C07299=1019.054,-103.989,386.792,-23.976,21.681,-44.335
C07300=1019.057,-103.662,386.769,-23.976,21.681,-44.331
C07301=1019.060,-103.334,386.746,-23.977,21.680,-44.326
C07302=1019.062,-103.008,386.723,-23.978,21.680,-44.320
C07303=1019.065,-102.682,386.701,-23.978,21.679,-44.316
C07304=1019.067,-102.357,386.678,-23.979,21.679,-44.311
C07305=1019.070,-102.032,386.656,-23.980,21.678,-44.307
C07306=1019.072,-101.707,386.634,-23.980,21.677,-44.302
C07307=1019.075,-101.383,386.610,-23.981,21.677,-44.298
C07308=1019.077,-101.059,386.588,-23.981,21.676,-44.292
C07309=1019.079,-100.736,386.565,-23.982,21.676,-44.287
C07310=1019.082,-100.413,386.543,-23.983,21.675,-44.283
C07311=1019.085,-100.091,386.520,-23.983,21.675,-44.278
C07312=1019.086,-99.770,386.498,-23.984,21.674,-44.274
C07313=1019.089,-99.448,386.475,-23.985,21.673,-44.268
C07314=1019.091,-99.127,386.453,-23.985,21.673,-44.265
C07315=1019.094,-98.805,386.430,-23.986,21.673,-44.260
C07316=1019.096,-98.484,386.408,-23.986,21.671,-44.255
C07317=1019.099,-98.163,386.385,-23.987,21.672,-44.250
C07318=1019.101,-97.843,386.363,-23.987,21.670,-44.246
C07319=1019.103,-97.521,386.340,-23.988,21.670,-44.241
C07320=1019.106,-97.201,386.317,-23.989,21.670,-44.236
C07321=1019.108,-96.880,386.295,-23.989,21.669,-44.231
C07322=1019.110,-96.559,386.273,-23.990,21.669,-44.226
C07323=1019.112,-96.237,386.251,-23.991,21.668,-44.222
C07324=1019.114,-95.916,386.227,-23.991,21.668,-44.217
C07325=1019.116,-95.594,386.206,-23.992,21.667,-44.213
C07326=1019.118,-95.272,386.183,-23.993,21.666,-44.207
C07327=1019.121,-94.949,386.159,-23.993,21.666,-44.204
C07328=1019.123,-94.626,386.137,-23.994,21.666,-44.199
C07329=1019.125,-94.303,386.114,-23.994,21.665,-44.193
C07330=1019.127,-93.978,386.091,-23.995,21.664,-44.189
C07331=1019.129,-93.654,386.068,-23.996,21.664,-44.184
C07332=1019.131,-93.329,386.045,-23.996,21.663,-44.180
C07333=1019.133,-93.003,386.022,-23.997,21.663,-44.175
C07334=1019.135,-92.676,385.999,-23.998,21.662,-44.169
C07335=1019.138,-92.350,385.976,-23.998,21.662,-44.165
C07336=1019.140,-92.022,385.953,-23.999,21.661,-44.160
C07337=1019.142,-91.695,385.930,-23.999,21.660,-44.156
C07338=1019.144,-91.367,385.907,-24.000,21.660,-44.150
C07339=1019.146,-91.038,385.883,-24.001,21.660,-44.145
C07340=1019.148,-90.709,385.859,-24.001,21.659,-44.141
C07341=1019.150,-90.380,385.836,-24.002,21.658,-44.136
C07342=1019.152,-90.041,385.812,-24.003,21.658,-44.130
C07343=1019.154,-89.635,385.783,-24.004,21.657,-44.123
C07344=1019.156,-89.404,385.767,-24.004,21.656,-44.121
C07345=1019.157,-89.166,385.750,-24.004,21.656,-44.119
C07346=1019.159,-88.933,385.733,-24.004,21.656,-44.117
C07347=1019.159,-88.714,385.718,-24.005,21.656,-44.114
C07348=1019.162,-88.342,385.691,-24.006,21.655,-44.106
C07349=1019.164,-88.024,385.668,-24.006,21.654,-44.102
C07350=1019.166,-87.711,385.646,-24.007,21.654,-44.097
C07351=1019.167,-87.400,385.624,-24.007,21.653,-44.093
C07352=1019.169,-87.088,385.602,-24.008,21.653,-44.088
C07353=1019.171,-86.771,385.579,-24.009,21.652,-44.082
C07354=1019.173,-86.449,385.556,-24.009,21.652,-44.078
C07355=1019.174,-86.120,385.532,-24.010,21.651,-44.073
C07356=1019.177,-85.760,385.507,-24.011,21.650,-44.067
C07357=1019.178,-85.352,385.478,-24.012,21.649,-44.062
C07358=1019.180,-85.138,385.462,-24.012,21.649,-44.060
C07359=1019.181,-84.926,385.447,-24.012,21.650,-44.056
C07360=1019.183,-84.528,385.418,-24.013,21.649,-44.051
C07361=1019.185,-84.179,385.393,-24.014,21.648,-44.045
C07362=1019.187,-83.845,385.369,-24.015,21.648,-44.040
C07363=1019.188,-83.510,385.345,-24.015,21.647,-44.036
C07364=1019.190,-83.175,385.321,-24.016,21.647,-44.031
C07365=1019.192,-82.839,385.297,-24.016,21.646,-44.025
C07366=1019.194,-82.503,385.273,-24.017,21.645,-44.021
C07367=1019.194,-82.166,385.249,-24.018,21.645,-44.016
C07368=1019.197,-81.830,385.224,-24.018,21.645,-44.010
C07369=1019.198,-81.492,385.200,-24.019,21.644,-44.005
C07370=1019.200,-81.155,385.176,-24.020,21.643,-44.001
C07371=1019.202,-80.816,385.151,-24.020,21.643,-43.995
C07372=1019.203,-80.477,385.127,-24.021,21.643,-43.990
C07373=1019.205,-80.139,385.102,-24.021,21.641,-43.986
C07374=1019.206,-79.799,385.077,-24.022,21.641,-43.981
C07375=1019.208,-79.459,385.053,-24.023,21.641,-43.975
C07376=1019.210,-79.119,385.029,-24.023,21.639,-43.971
C07377=1019.211,-78.779,385.004,-24.024,21.639,-43.966
C07378=1019.212,-78.438,384.979,-24.025,21.638,-43.960
C07379=1019.214,-78.097,384.954,-24.026,21.639,-43.955
C07380=1019.215,-77.755,384.930,-24.026,21.637,-43.951
C07381=1019.217,-77.414,384.905,-24.027,21.637,-43.946
C07382=1019.218,-77.072,384.879,-24.028,21.636,-43.940
C07383=1019.220,-76.730,384.855,-24.028,21.636,-43.936
C07384=1019.221,-76.387,384.830,-24.029,21.635,-43.931
C07385=1019.223,-76.045,384.805,-24.030,21.635,-43.926
C07386=1019.224,-75.702,384.780,-24.030,21.634,-43.920
C07387=1019.225,-75.358,384.755,-24.031,21.634,-43.916
C07388=1019.226,-75.015,384.730,-24.031,21.633,-43.911
C07389=1019.228,-74.672,384.705,-24.032,21.633,-43.905
C07390=1019.230,-74.329,384.680,-24.033,21.632,-43.901
C07391=1019.231,-73.984,384.655,-24.033,21.632,-43.896
C07392=1019.232,-73.641,384.630,-24.034,21.631,-43.890
C07393=1019.233,-73.297,384.604,-24.035,21.630,-43.885
C07394=1019.235,-72.954,384.578,-24.035,21.630,-43.881
C07395=1019.236,-72.609,384.554,-24.036,21.629,-43.875
C07396=1019.237,-72.266,384.529,-24.037,21.629,-43.870
C07397=1019.238,-71.921,384.504,-24.038,21.628,-43.865
C07398=1019.240,-71.578,384.478,-24.038,21.628,-43.861
C07399=1019.241,-71.233,384.453,-24.039,21.627,-43.855
C07400=1019.242,-70.889,384.428,-24.040,21.627,-43.850
C07401=1019.243,-70.545,384.402,-24.040,21.626,-43.844
C07402=1019.244,-70.202,384.377,-24.041,21.625,-43.840
C07403=1019.246,-69.858,384.352,-24.041,21.625,-43.835
C07404=1019.246,-69.513,384.327,-24.042,21.624,-43.829
C07405=1019.248,-69.169,384.301,-24.043,21.624,-43.824
C07406=1019.249,-68.825,384.275,-24.043,21.623,-43.820
C07407=1019.249,-68.482,384.251,-24.044,21.623,-43.815
C07408=1019.251,-68.138,384.225,-24.045,21.622,-43.809
C07409=1019.252,-67.795,384.200,-24.045,21.622,-43.805
C07410=1019.253,-67.451,384.174,-24.046,21.621,-43.800
C07411=1019.254,-67.108,384.149,-24.047,21.621,-43.795
C07412=1019.255,-66.764,384.124,-24.048,21.620,-43.789
C07413=1019.256,-66.422,384.098,-24.048,21.620,-43.785
C07414=1019.257,-66.079,384.073,-24.049,21.619,-43.780
C07415=1019.258,-65.736,384.047,-24.050,21.619,-43.774
C07416=1019.259,-65.394,384.022,-24.050,21.617,-43.770
C07417=1019.260,-65.051,383.996,-24.051,21.618,-43.765
C07418=1019.261,-64.710,383.971,-24.051,21.617,-43.759
C07419=1019.262,-64.368,383.946,-24.052,21.617,-43.754
C07420=1019.262,-64.027,383.921,-24.053,21.615,-43.750
C07421=1019.264,-63.686,383.895,-24.053,21.616,-43.745
C07422=1019.264,-63.346,383.870,-24.054,21.615,-43.739
C07423=1019.265,-63.005,383.845,-24.055,21.614,-43.735
C07424=1019.266,-62.665,383.819,-24.055,21.613,-43.730
C07425=1019.266,-62.326,383.794,-24.056,21.614,-43.725
C07426=1019.267,-61.987,383.769,-24.057,21.612,-43.720
C07427=1019.268,-61.648,383.743,-24.057,21.612,-43.715
C07428=1019.269,-61.309,383.718,-24.058,21.611,-43.710
C07429=1019.270,-60.972,383.693,-24.059,21.611,-43.706
C07430=1019.270,-60.633,383.667,-24.059,21.610,-43.700
C07431=1019.271,-60.296,383.642,-24.060,21.610,-43.695
C07432=1019.272,-59.960,383.617,-24.060,21.609,-43.691
C07433=1019.272,-59.623,383.592,-24.061,21.609,-43.686
C07434=1019.272,-59.287,383.567,-24.062,21.608,-43.680
C07435=1019.274,-58.951,383.541,-24.062,21.608,-43.676
C07436=1019.274,-58.616,383.516,-24.063,21.607,-43.671
C07437=1019.275,-58.281,383.491,-24.064,21.607,-43.666
C07438=1019.276,-57.946,383.466,-24.064,21.606,-43.662
C07439=1019.276,-57.612,383.441,-24.065,21.606,-43.656
C07440=1019.276,-57.279,383.416,-24.066,21.605,-43.652
C07441=1019.277,-56.945,383.390,-24.066,21.604,-43.647
C07442=1019.277,-56.612,383.365,-24.067,21.605,-43.642
C07443=1019.279,-56.278,383.340,-24.068,21.603,-43.637
C07444=1019.278,-55.946,383.315,-24.068,21.603,-43.632
C07445=1019.279,-55.612,383.290,-24.069,21.603,-43.627
C07446=1019.280,-55.280,383.265,-24.070,21.602,-43.623
C07447=1019.280,-54.947,383.240,-24.070,21.602,-43.618
C07448=1019.281,-54.615,383.215,-24.071,21.601,-43.613
C07449=1019.281,-54.283,383.190,-24.072,21.601,-43.608
C07450=1019.281,-53.950,383.164,-24.072,21.600,-43.603
C07451=1019.282,-53.618,383.140,-24.073,21.599,-43.599
C07452=1019.282,-53.286,383.114,-24.074,21.600,-43.594
C07453=1019.283,-52.953,383.090,-24.074,21.598,-43.589
C07454=1019.283,-52.621,383.064,-24.075,21.598,-43.584
C07455=1019.283,-52.289,383.038,-24.075,21.597,-43.579
C07456=1019.284,-51.956,383.014,-24.076,21.597,-43.575
C07457=1019.284,-51.624,382.988,-24.077,21.597,-43.570
C07458=1019.284,-51.292,382.963,-24.077,21.596,-43.566
C07459=1019.285,-50.959,382.938,-24.078,21.596,-43.560
C07460=1019.285,-50.627,382.912,-24.079,21.595,-43.555
C07461=1019.285,-50.295,382.887,-24.079,21.594,-43.551
C07462=1019.285,-49.962,382.862,-24.080,21.595,-43.546
C07463=1019.285,-49.630,382.836,-24.080,21.593,-43.542
C07464=1019.286,-49.297,382.812,-24.081,21.593,-43.536
C07465=1019.286,-48.965,382.786,-24.081,21.592,-43.532
C07466=1019.287,-48.633,382.760,-24.082,21.592,-43.527
C07467=1019.286,-48.300,382.735,-24.083,21.592,-43.522
C07468=1019.287,-47.968,382.710,-24.083,21.591,-43.518
C07469=1019.287,-47.635,382.685,-24.084,21.591,-43.512
C07470=1019.287,-47.303,382.659,-24.085,21.589,-43.508
C07471=1019.287,-46.971,382.633,-24.086,21.589,-43.503
C07472=1019.287,-46.638,382.608,-24.086,21.590,-43.498
C07473=1019.287,-46.306,382.583,-24.087,21.588,-43.494
C07474=1019.287,-45.973,382.558,-24.088,21.588,-43.488
C07475=1019.287,-45.641,382.532,-24.088,21.588,-43.485
C07476=1019.288,-45.309,382.506,-24.089,21.587,-43.479
C07477=1019.287,-44.975,382.481,-24.089,21.586,-43.475
C07478=1019.288,-44.642,382.455,-24.090,21.586,-43.470
C07479=1019.288,-44.310,382.430,-24.091,21.586,-43.465
C07480=1019.288,-43.977,382.404,-24.091,21.585,-43.461
C07481=1019.288,-43.645,382.378,-24.092,21.585,-43.455
C07482=1019.287,-43.312,382.353,-24.092,21.584,-43.451
C07483=1019.287,-42.980,382.327,-24.093,21.583,-43.446
C07484=1019.288,-42.648,382.301,-24.094,21.583,-43.442
C07485=1019.288,-42.315,382.276,-24.094,21.583,-43.437
C07486=1019.287,-41.982,382.250,-24.095,21.582,-43.431
C07487=1019.287,-41.650,382.225,-24.096,21.582,-43.427
C07488=1019.286,-41.317,382.199,-24.096,21.582,-43.422
C07489=1019.287,-40.985,382.173,-24.097,21.580,-43.418
C07490=1019.287,-40.652,382.148,-24.098,21.580,-43.413
C07491=1019.287,-40.319,382.122,-24.098,21.580,-43.409
C07492=1019.287,-39.987,382.096,-24.099,21.579,-43.404
C07493=1019.286,-39.653,382.070,-24.100,21.579,-43.398
C07494=1019.286,-39.321,382.045,-24.100,21.578,-43.394
C07495=1019.286,-38.989,382.018,-24.101,21.578,-43.389
C07496=1019.286,-38.656,381.993,-24.101,21.577,-43.385
C07497=1019.285,-38.323,381.967,-24.102,21.577,-43.380
C07498=1019.285,-37.991,381.941,-24.102,21.576,-43.376
C07499=1019.285,-37.658,381.916,-24.103,21.576,-43.371
C07500=1019.285,-37.326,381.890,-24.104,21.575,-43.366
C07501=1019.284,-36.993,381.864,-24.105,21.575,-43.361
C07502=1019.284,-36.659,381.838,-24.105,21.574,-43.357
C07503=1019.284,-36.327,381.812,-24.106,21.574,-43.352
C07504=1019.284,-35.995,381.786,-24.107,21.574,-43.347
C07505=1019.283,-35.662,381.760,-24.107,21.573,-43.343
C07506=1019.283,-35.329,381.734,-24.108,21.573,-43.337
C07507=1019.283,-34.997,381.708,-24.108,21.572,-43.334
C07508=1019.282,-34.664,381.682,-24.109,21.572,-43.328
C07509=1019.281,-34.331,381.657,-24.109,21.571,-43.324
C07510=1019.281,-33.999,381.630,-24.110,21.571,-43.319
C07511=1019.281,-33.667,381.605,-24.111,21.570,-43.315
C07512=1019.280,-33.333,381.579,-24.111,21.570,-43.310
C07513=1019.280,-33.000,381.552,-24.112,21.569,-43.306
C07514=1019.280,-32.668,381.526,-24.113,21.569,-43.301
C07515=1019.279,-32.335,381.500,-24.113,21.568,-43.296
C07516=1019.279,-32.002,381.474,-24.114,21.568,-43.291
C07517=1019.278,-31.669,381.448,-24.114,21.567,-43.287
C07518=1019.278,-31.337,381.422,-24.115,21.567,-43.282
C07519=1019.277,-31.004,381.396,-24.116,21.566,-43.278
C07520=1019.276,-30.671,381.370,-24.116,21.566,-43.273
C07521=1019.276,-30.339,381.344,-24.117,21.565,-43.269
C07522=1019.275,-30.006,381.317,-24.118,21.565,-43.264
C07523=1019.274,-29.673,381.292,-24.118,21.565,-43.260
C07524=1019.275,-29.340,381.265,-24.119,21.564,-43.254
C07525=1019.274,-29.007,381.239,-24.119,21.563,-43.250
C07526=1019.273,-28.675,381.212,-24.120,21.563,-43.245
C07527=1019.273,-28.342,381.186,-24.120,21.562,-43.241
C07528=1019.272,-28.009,381.161,-24.121,21.562,-43.236
C07529=1019.271,-27.676,381.134,-24.122,21.562,-43.232
C07530=1019.270,-27.344,381.107,-24.123,21.562,-43.227
C07531=1019.270,-27.011,381.081,-24.123,21.560,-43.223
C07532=1019.269,-26.678,381.056,-24.124,21.560,-43.217
C07533=1019.269,-26.346,381.029,-24.124,21.560,-43.214
C07534=1019.267,-26.013,381.002,-24.125,21.559,-43.208
C07535=1019.267,-25.680,380.976,-24.126,21.559,-43.204
C07536=1019.266,-25.348,380.950,-24.126,21.559,-43.199
C07537=1019.265,-25.014,380.923,-24.127,21.558,-43.195
C07538=1019.265,-24.681,380.897,-24.128,21.558,-43.190
C07539=1019.264,-24.349,380.871,-24.128,21.557,-43.186
C07540=1019.263,-24.016,380.844,-24.129,21.557,-43.181
C07541=1019.263,-23.683,380.818,-24.129,21.556,-43.177
C07542=1019.262,-23.351,380.791,-24.130,21.556,-43.171
C07543=1019.260,-23.017,380.765,-24.131,21.555,-43.168
C07544=1019.260,-22.685,380.739,-24.131,21.556,-43.162
C07545=1019.259,-22.352,380.712,-24.132,21.554,-43.158
C07546=1019.258,-22.019,380.686,-24.133,21.554,-43.153
C07547=1019.257,-21.687,380.659,-24.133,21.554,-43.149
C07548=1019.256,-21.354,380.633,-24.134,21.553,-43.144
C07549=1019.255,-21.021,380.606,-24.134,21.552,-43.140
C07550=1019.254,-20.688,380.580,-24.135,21.553,-43.135
C07551=1019.253,-20.355,380.553,-24.136,21.552,-43.131
C07552=1019.253,-20.023,380.527,-24.136,21.551,-43.127
C07553=1019.251,-19.690,380.500,-24.137,21.551,-43.122
C07554=1019.251,-19.517,380.486,-24.137,21.550,-43.118
C07555=1019.250,-19.101,380.453,-24.138,21.550,-43.112
C07556=1019.249,-18.853,380.433,-24.139,21.550,-43.109
C07557=1019.248,-18.591,380.411,-24.139,21.550,-43.107
C07558=1019.248,-18.329,380.391,-24.139,21.549,-43.105
C07559=1019.247,-18.082,380.371,-24.139,21.548,-43.103
C07560=1019.246,-17.860,380.353,-24.140,21.549,-43.100
C07561=1019.245,-17.495,380.324,-24.141,21.548,-43.092
C07562=1019.244,-17.163,380.297,-24.141,21.547,-43.088
C07563=1019.243,-16.829,380.271,-24.142,21.547,-43.083
C07564=1019.241,-16.496,380.244,-24.142,21.547,-43.079
C07565=1019.240,-16.162,380.218,-24.143,21.546,-43.074
C07566=1019.240,-15.829,380.190,-24.144,21.546,-43.070
C07567=1019.238,-15.493,380.164,-24.145,21.546,-43.065
C07568=1019.237,-15.157,380.137,-24.145,21.545,-43.061
C07569=1019.236,-14.819,380.109,-24.146,21.544,-43.055
C07570=1019.235,-14.478,380.082,-24.146,21.544,-43.052
C07571=1019.233,-14.137,380.054,-24.147,21.544,-43.046
C07572=1019.232,-13.792,380.027,-24.147,21.543,-43.042
C07573=1019.231,-13.445,379.999,-24.148,21.543,-43.037
C07574=1019.230,-13.098,379.971,-24.149,21.542,-43.033
C07575=1019.228,-12.747,379.943,-24.149,21.542,-43.028
C07576=1019.227,-12.395,379.914,-24.150,21.541,-43.024
C07577=1019.226,-12.042,379.885,-24.151,21.541,-43.019
C07578=1019.224,-11.687,379.857,-24.151,21.540,-43.014
C07579=1019.223,-11.330,379.829,-24.152,21.540,-43.009
C07580=1019.222,-10.972,379.800,-24.152,21.539,-43.006
C07581=1019.220,-10.613,379.770,-24.153,21.539,-43.000
C07582=1019.219,-10.254,379.741,-24.154,21.539,-42.995
C07583=1019.217,-9.893,379.711,-24.154,21.538,-42.991
C07584=1019.216,-9.532,379.682,-24.155,21.538,-42.985
C07585=1019.215,-9.169,379.653,-24.156,21.537,-42.982
C07586=1019.213,-8.806,379.624,-24.156,21.536,-42.976
C07587=1019.212,-8.444,379.594,-24.157,21.536,-42.971
C07588=1019.210,-8.081,379.564,-24.158,21.536,-42.967
C07589=1019.208,-7.717,379.536,-24.158,21.535,-42.961
C07590=1019.206,-7.351,379.505,-24.159,21.535,-42.956
C07591=1019.205,-6.983,379.476,-24.160,21.534,-42.952
C07592=1019.203,-6.611,379.445,-24.160,21.534,-42.947
C07593=1019.201,-6.236,379.414,-24.161,21.533,-42.941
C07594=1019.199,-5.861,379.384,-24.162,21.533,-42.937
C07595=1019.198,-5.485,379.353,-24.163,21.533,-42.932
C07596=1019.196,-5.111,379.323,-24.163,21.532,-42.928
C07597=1019.194,-4.741,379.293,-24.164,21.532,-42.923
C07598=1019.193,-4.375,379.263,-24.164,21.531,-42.919
C07599=1019.191,-4.014,379.233,-24.165,21.530,-42.913
C07600=1019.189,-3.656,379.204,-24.166,21.531,-42.908
C07601=1019.187,-3.302,379.175,-24.166,21.529,-42.904
C07602=1019.186,-2.950,379.147,-24.167,21.529,-42.899
C07603=1019.184,-2.598,379.118,-24.167,21.529,-42.895
C07604=1019.183,-2.249,379.089,-24.168,21.529,-42.890
C07605=1019.181,-1.899,379.060,-24.169,21.528,-42.886
C07606=1019.179,-1.553,379.032,-24.169,21.528,-42.880
C07607=1019.177,-1.208,379.004,-24.170,21.527,-42.877
C07608=1019.175,-0.865,378.976,-24.170,21.527,-42.873
C07609=1019.174,-0.523,378.947,-24.171,21.526,-42.867
C07610=1019.172,-0.183,378.920,-24.172,21.526,-42.864
C07611=1019.170,0.155,378.892,-24.172,21.526,-42.858
C07612=1019.168,0.493,378.865,-24.173,21.525,-42.855
C07613=1019.166,0.828,378.837,-24.173,21.525,-42.851
C07614=1019.165,1.164,378.809,-24.174,21.525,-42.846
C07615=1019.163,1.497,378.782,-24.175,21.524,-42.842
C07616=1019.161,1.831,378.754,-24.175,21.523,-42.838
C07617=1019.160,2.161,378.727,-24.176,21.523,-42.834
C07618=1019.158,2.474,378.701,-24.176,21.523,-42.831
C07619=1019.155,2.762,378.678,-24.177,21.522,-42.827
C07620=1019.154,3.031,378.655,-24.177,21.522,-42.823
C07621=1019.152,3.292,378.633,-24.178,21.522,-42.818
C07622=1019.152,3.563,378.611,-24.179,21.521,-42.814
C07623=1019.150,3.852,378.588,-24.179,21.521,-42.810
C07624=1019.148,4.165,378.562,-24.179,21.520,-42.807
C07625=1019.146,4.495,378.535,-24.180,21.521,-42.803
C07626=1019.144,4.826,378.508,-24.180,21.519,-42.799
C07627=1019.142,5.157,378.479,-24.181,21.519,-42.795
C07628=1019.140,5.488,378.452,-24.181,21.518,-42.792
C07629=1019.139,5.818,378.425,-24.182,21.519,-42.786
C07630=1019.136,6.148,378.397,-24.183,21.518,-42.783
C07631=1019.135,6.478,378.370,-24.183,21.518,-42.779
C07632=1019.133,6.807,378.343,-24.184,21.518,-42.774
C07633=1019.131,7.135,378.316,-24.185,21.517,-42.770
C07634=1019.129,7.463,378.289,-24.185,21.517,-42.766
C07635=1019.126,7.788,378.262,-24.186,21.516,-42.762
C07636=1019.125,8.111,378.235,-24.186,21.516,-42.759
C07637=1019.122,8.432,378.208,-24.186,21.515,-42.755
C07638=1019.121,8.750,378.182,-24.187,21.516,-42.750
C07639=1019.119,9.067,378.156,-24.188,21.515,-42.746
C07640=1019.116,9.382,378.130,-24.188,21.515,-42.742
C07641=1019.115,9.697,378.104,-24.189,21.514,-42.738
C07642=1019.112,10.011,378.077,-24.190,21.514,-42.733
C07643=1019.110,10.327,378.051,-24.190,21.514,-42.730
C07644=1019.108,10.644,378.025,-24.191,21.513,-42.726
C07645=1019.106,10.963,377.998,-24.191,21.513,-42.722
C07646=1019.104,11.283,377.971,-24.192,21.512,-42.718
C07647=1019.102,11.605,377.944,-24.192,21.512,-42.715
C07648=1019.100,11.929,377.917,-24.193,21.511,-42.711
C07649=1019.098,12.253,377.891,-24.193,21.511,-42.707
C07650=1019.096,12.576,377.864,-24.194,21.511,-42.702
C07651=1019.093,12.899,377.836,-24.194,21.510,-42.698
C07652=1019.091,13.223,377.810,-24.195,21.510,-42.694
C07653=1019.089,13.547,377.782,-24.195,21.509,-42.691
C07654=1019.087,13.871,377.755,-24.196,21.509,-42.687
C07655=1019.084,14.195,377.729,-24.197,21.509,-42.682
C07656=1019.083,14.520,377.702,-24.197,21.509,-42.678
C07657=1019.080,14.845,377.674,-24.198,21.508,-42.674
C07658=1019.077,15.171,377.647,-24.198,21.508,-42.670
C07659=1019.076,15.496,377.620,-24.199,21.507,-42.667
C07660=1019.074,15.823,377.592,-24.199,21.507,-42.663
C07661=1019.070,16.150,377.565,-24.200,21.507,-42.658
C07662=1019.069,16.477,377.537,-24.200,21.506,-42.654
C07663=1019.066,16.805,377.510,-24.201,21.506,-42.650
C07664=1019.064,17.134,377.482,-24.201,21.505,-42.646
C07665=1019.061,17.464,377.455,-24.202,21.505,-42.643
C07666=1019.059,17.793,377.427,-24.202,21.504,-42.639
C07667=1019.056,18.124,377.399,-24.203,21.504,-42.634
C07668=1019.054,18.454,377.371,-24.204,21.504,-42.630
C07669=1019.051,18.786,377.343,-24.204,21.503,-42.626
C07670=1019.049,19.118,377.315,-24.205,21.503,-42.622
C07671=1019.047,19.449,377.288,-24.205,21.502,-42.619
C07672=1019.044,19.798,377.258,-24.206,21.503,-42.613
C07673=1019.041,20.215,377.223,-24.207,21.502,-42.608
C07674=1019.039,20.451,377.204,-24.207,21.502,-42.604
C07675=1019.037,20.698,377.182,-24.207,21.502,-42.603
C07676=1019.035,20.946,377.162,-24.208,21.502,-42.601
C07677=1019.033,21.188,377.141,-24.208,21.502,-42.599
C07678=1019.031,21.415,377.123,-24.208,21.501,-42.597
C07679=1019.029,21.622,377.105,-24.209,21.501,-42.593
C07680=1019.027,21.979,377.075,-24.209,21.500,-42.588
C07681=1019.025,22.303,377.047,-24.210,21.501,-42.584
C07682=1019.022,22.597,377.022,-24.210,21.500,-42.582
C07683=1019.020,22.850,377.001,-24.210,21.499,-42.580
C07684=1019.017,23.260,376.966,-24.211,21.499,-42.573
C07685=1019.014,23.668,376.932,-24.212,21.498,-42.565
C07686=1019.012,23.920,376.910,-24.213,21.498,-42.562
C07687=1019.009,24.214,376.886,-24.213,21.498,-42.560
C07688=1019.006,24.541,376.858,-24.213,21.497,-42.558
C07689=1019.004,24.875,376.830,-24.214,21.497,-42.553
C07690=1019.001,25.209,376.801,-24.215,21.497,-42.549
C07691=1018.998,25.544,376.773,-24.215,21.496,-42.545
C07692=1018.996,25.878,376.745,-24.216,21.496,-42.541
C07693=1018.992,26.212,376.717,-24.216,21.495,-42.538
C07694=1018.990,26.546,376.689,-24.217,21.495,-42.534
C07695=1018.987,26.881,376.659,-24.217,21.494,-42.530
C07696=1018.985,27.216,376.632,-24.218,21.494,-42.525
C07697=1018.982,27.549,376.603,-24.219,21.495,-42.522
C07698=1018.979,27.884,376.574,-24.219,21.494,-42.518
C07699=1018.976,28.219,376.546,-24.220,21.494,-42.514
C07700=1018.973,28.553,376.518,-24.220,21.493,-42.510
C07701=1018.970,28.887,376.490,-24.221,21.493,-42.507
C07702=1018.967,29.222,376.461,-24.221,21.492,-42.503
C07703=1018.965,29.556,376.432,-24.222,21.493,-42.498
C07704=1018.961,29.891,376.404,-24.222,21.492,-42.494
C07705=1018.959,30.225,376.376,-24.223,21.492,-42.490
C07706=1018.955,30.560,376.347,-24.223,21.491,-42.486
C07707=1018.953,30.895,376.318,-24.224,21.491,-42.483
C07708=1018.949,31.229,376.290,-24.224,21.490,-42.479
C07709=1018.947,31.563,376.262,-24.225,21.490,-42.475
C07710=1018.944,31.898,376.233,-24.225,21.489,-42.471
C07711=1018.941,32.233,376.204,-24.226,21.489,-42.468
C07712=1018.938,32.567,376.175,-24.226,21.489,-42.464
C07713=1018.934,32.902,376.147,-24.227,21.489,-42.459
C07714=1018.931,33.236,376.118,-24.228,21.489,-42.455
C07715=1018.928,33.571,376.090,-24.228,21.488,-42.452
C07716=1018.925,33.906,376.061,-24.229,21.488,-42.448
C07717=1018.922,34.241,376.033,-24.229,21.487,-42.444
C07718=1018.919,34.574,376.005,-24.230,21.487,-42.440
C07719=1018.916,34.909,375.976,-24.230,21.486,-42.437
C07720=1018.912,35.244,375.947,-24.231,21.486,-42.433
C07721=1018.910,35.579,375.918,-24.231,21.485,-42.429
C07722=1018.906,35.914,375.889,-24.232,21.486,-42.426
C07723=1018.903,36.248,375.861,-24.232,21.485,-42.422
C07724=1018.900,36.583,375.832,-24.233,21.485,-42.418
C07725=1018.897,36.917,375.803,-24.234,21.485,-42.413
C07726=1018.894,37.252,375.775,-24.234,21.485,-42.409
C07727=1018.891,37.587,375.746,-24.235,21.484,-42.405
C07728=1018.888,37.922,375.718,-24.235,21.484,-42.402
C07729=1018.884,38.257,375.688,-24.236,21.483,-42.398
C07730=1018.880,38.591,375.660,-24.236,21.483,-42.395
C07731=1018.877,38.926,375.631,-24.237,21.483,-42.391
C07732=1018.874,39.261,375.603,-24.237,21.483,-42.387
C07733=1018.871,39.596,375.573,-24.238,21.482,-42.383
C07734=1018.867,39.931,375.545,-24.238,21.482,-42.380
C07735=1018.865,40.265,375.516,-24.239,21.481,-42.376
C07736=1018.860,40.600,375.487,-24.239,21.481,-42.372
C07737=1018.857,40.934,375.458,-24.240,21.481,-42.369
C07738=1018.854,41.269,375.430,-24.240,21.481,-42.365
C07739=1018.850,41.604,375.400,-24.241,21.480,-42.361
C07740=1018.847,41.939,375.372,-24.241,21.480,-42.357
C07741=1018.844,42.274,375.344,-24.242,21.479,-42.354
C07742=1018.840,42.609,375.314,-24.242,21.479,-42.350
C07743=1018.837,42.944,375.286,-24.243,21.479,-42.347
C07744=1018.833,43.278,375.257,-24.243,21.479,-42.343
C07745=1018.830,43.614,375.228,-24.244,21.478,-42.339
C07746=1018.826,43.948,375.199,-24.244,21.478,-42.335
C07747=1018.823,44.284,375.170,-24.245,21.477,-42.332
C07748=1018.820,44.618,375.141,-24.245,21.477,-42.328
C07749=1018.816,44.953,375.112,-24.246,21.477,-42.325
C07750=1018.813,45.288,375.083,-24.246,21.477,-42.321
C07751=1018.809,45.624,375.054,-24.247,21.476,-42.317
C07752=1018.805,45.957,375.025,-24.247,21.476,-42.313
C07753=1018.801,46.293,374.996,-24.248,21.475,-42.309
C07754=1018.798,46.628,374.967,-24.248,21.475,-42.306
C07755=1018.795,46.963,374.938,-24.249,21.475,-42.302
C07756=1018.791,47.298,374.909,-24.249,21.475,-42.299
C07757=1018.787,47.633,374.880,-24.250,21.474,-42.295
C07758=1018.784,47.968,374.851,-24.250,21.474,-42.291
C07759=1018.780,48.302,374.822,-24.251,21.473,-42.287
C07760=1018.776,48.638,374.793,-24.251,21.473,-42.284
C07761=1018.772,48.973,374.764,-24.252,21.473,-42.280
C07762=1018.769,49.308,374.735,-24.252,21.473,-42.277
C07763=1018.765,49.642,374.706,-24.253,21.472,-42.273
C07764=1018.762,49.978,374.677,-24.253,21.472,-42.269
C07765=1018.758,50.313,374.647,-24.254,21.472,-42.266
C07766=1018.753,50.647,374.619,-24.254,21.471,-42.262
C07767=1018.750,50.983,374.590,-24.255,21.471,-42.258
C07768=1018.747,51.317,374.561,-24.255,21.471,-42.254
C07769=1018.743,51.653,374.532,-24.256,21.471,-42.251
C07770=1018.739,51.988,374.502,-24.256,21.470,-42.247
C07771=1018.735,52.323,374.473,-24.257,21.470,-42.244
C07772=1018.731,52.657,374.444,-24.257,21.470,-42.240
C07773=1018.727,52.993,374.415,-24.258,21.469,-42.238
C07774=1018.723,53.327,374.385,-24.258,21.469,-42.234
C07775=1018.720,53.663,374.357,-24.259,21.468,-42.230
C07776=1018.716,53.998,374.327,-24.259,21.468,-42.227
C07777=1018.711,54.332,374.298,-24.260,21.468,-42.223
C07778=1018.708,54.667,374.269,-24.260,21.468,-42.220
C07779=1018.704,55.003,374.240,-24.261,21.467,-42.216
C07780=1018.700,55.338,374.211,-24.261,21.467,-42.212
C07781=1018.696,55.673,374.181,-24.262,21.467,-42.209
C07782=1018.691,56.008,374.152,-24.262,21.467,-42.205
C07783=1018.688,56.343,374.123,-24.263,21.466,-42.201
C07784=1018.684,56.678,374.094,-24.263,21.466,-42.197
C07785=1018.680,57.013,374.064,-24.264,21.466,-42.194
C07786=1018.676,57.348,374.035,-24.264,21.465,-42.192
C07787=1018.672,57.682,374.006,-24.264,21.465,-42.188
C07788=1018.668,58.018,373.977,-24.265,21.464,-42.184
C07789=1018.664,58.353,373.947,-24.266,21.465,-42.181
C07790=1018.660,58.688,373.918,-24.266,21.464,-42.177
C07791=1018.656,59.022,373.889,-24.267,21.464,-42.173
C07792=1018.652,59.358,373.860,-24.267,21.464,-42.170
C07793=1018.647,59.693,373.829,-24.268,21.464,-42.166
C07794=1018.643,60.028,373.801,-24.268,21.463,-42.163
C07795=1018.639,60.363,373.771,-24.268,21.462,-42.160
C07796=1018.634,60.698,373.742,-24.269,21.462,-42.157
C07797=1018.631,61.033,373.712,-24.269,21.462,-42.153
C07798=1018.626,61.368,373.684,-24.270,21.461,-42.149
C07799=1018.622,61.703,373.653,-24.270,21.462,-42.146
C07800=1018.618,62.038,373.624,-24.271,21.461,-42.142
C07801=1018.614,62.372,373.595,-24.271,21.461,-42.139
C07802=1018.610,62.710,373.566,-24.272,21.460,-42.135
C07803=1018.604,63.106,373.531,-24.272,21.460,-42.131
C07804=1018.601,63.329,373.511,-24.273,21.461,-42.130
C07805=1018.600,63.547,373.491,-24.273,21.460,-42.128
C07806=1018.599,63.921,373.456,-24.274,21.460,-42.124
C07807=1018.598,64.278,373.423,-24.274,21.459,-42.120
C07808=1018.597,64.663,373.386,-24.274,21.459,-42.116
C07809=1018.596,65.059,373.349,-24.275,21.458,-42.113
C07810=1018.594,65.436,373.314,-24.276,21.459,-42.108
C07811=1018.594,65.790,373.280,-24.276,21.457,-42.105
C07812=1018.593,66.129,373.248,-24.277,21.458,-42.102
C07813=1018.592,66.462,373.216,-24.277,21.457,-42.098
C07814=1018.591,66.797,373.185,-24.278,21.457,-42.094
C07815=1018.590,67.134,373.153,-24.278,21.457,-42.091
C07816=1018.589,67.473,373.122,-24.279,21.457,-42.087
C07817=1018.588,67.811,373.089,-24.279,21.456,-42.085
C07818=1018.587,68.150,373.058,-24.279,21.456,-42.082
C07819=1018.587,68.490,373.025,-24.280,21.456,-42.078
C07820=1018.585,68.832,372.993,-24.280,21.455,-42.074
C07821=1018.584,69.173,372.960,-24.281,21.456,-42.071
C07822=1018.583,69.516,372.928,-24.281,21.455,-42.067
C07823=1018.582,69.860,372.896,-24.282,21.455,-42.063
C07824=1018.581,70.205,372.863,-24.282,21.454,-42.061
C07825=1018.580,70.550,372.830,-24.283,21.454,-42.058
C07826=1018.579,70.894,372.797,-24.283,21.453,-42.054
C07827=1018.578,71.238,372.765,-24.284,21.454,-42.051
C07828=1018.577,71.583,372.732,-24.284,21.453,-42.047
C07829=1018.576,71.928,372.699,-24.285,21.453,-42.043
C07830=1018.575,72.273,372.667,-24.285,21.453,-42.041
C07831=1018.574,72.619,372.633,-24.285,21.452,-42.037
C07832=1018.573,72.967,372.601,-24.286,21.452,-42.034
C07833=1018.572,73.317,372.567,-24.286,21.451,-42.030
C07834=1018.571,73.669,372.533,-24.287,21.452,-42.027
C07835=1018.570,74.022,372.500,-24.288,21.451,-42.023
C07836=1018.569,74.377,372.467,-24.288,21.451,-42.019
C07837=1018.568,74.734,372.432,-24.288,21.451,-42.017
C07838=1018.567,75.092,372.398,-24.289,21.450,-42.013
C07839=1018.566,75.449,372.364,-24.289,21.450,-42.010
C07840=1018.564,75.804,372.330,-24.290,21.450,-42.006
C07841=1018.563,76.151,372.297,-24.290,21.449,-42.004
C07842=1018.562,76.494,372.264,-24.291,21.449,-42.001
C07843=1018.562,76.830,372.232,-24.291,21.449,-41.997
C07844=1018.561,77.161,372.201,-24.292,21.449,-41.994
C07845=1018.559,77.487,372.169,-24.292,21.449,-41.990
C07846=1018.558,77.810,372.138,-24.292,21.448,-41.987
C07847=1018.558,78.134,372.108,-24.293,21.448,-41.984
C07848=1018.557,78.458,372.076,-24.293,21.448,-41.980
C07849=1018.555,78.786,372.045,-24.294,21.447,-41.977
C07850=1018.554,79.119,372.012,-24.295,21.448,-41.973
C07851=1018.553,79.457,371.980,-24.295,21.446,-41.971
C07852=1018.553,79.803,371.947,-24.295,21.447,-41.968
C07853=1018.551,80.154,371.914,-24.296,21.446,-41.964
C07854=1018.551,80.509,371.879,-24.296,21.446,-41.962
C07855=1018.549,80.865,371.845,-24.297,21.446,-41.958
C07856=1018.548,81.222,371.811,-24.297,21.445,-41.955
C07857=1018.546,81.578,371.776,-24.298,21.446,-41.951
C07858=1018.545,81.934,371.743,-24.298,21.445,-41.947
C07859=1018.544,82.288,371.708,-24.298,21.444,-41.945
C07860=1018.543,82.642,371.674,-24.299,21.444,-41.942
C07861=1018.542,82.995,371.641,-24.299,21.444,-41.938
C07862=1018.541,83.346,371.606,-24.300,21.444,-41.935
C07863=1018.540,83.697,371.573,-24.300,21.444,-41.931
C07864=1018.538,84.048,371.539,-24.301,21.443,-41.929
C07865=1018.537,84.396,371.505,-24.301,21.443,-41.925
C07866=1018.536,84.744,371.471,-24.302,21.443,-41.922
C07867=1018.536,85.091,371.438,-24.302,21.443,-41.918
C07868=1018.534,85.436,371.405,-24.302,21.442,-41.916
C07869=1018.534,85.780,371.371,-24.303,21.442,-41.912
C07870=1018.532,86.123,371.339,-24.303,21.442,-41.909
C07871=1018.531,86.465,371.305,-24.304,21.441,-41.906
C07872=1018.529,86.806,371.272,-24.304,21.441,-41.903
C07873=1018.529,87.146,371.240,-24.305,21.441,-41.899
C07874=1018.527,87.482,371.207,-24.305,21.441,-41.898
C07875=1018.526,87.815,371.174,-24.305,21.440,-41.894
C07876=1018.525,88.142,371.143,-24.306,21.441,-41.890
C07877=1018.524,88.464,371.112,-24.306,21.439,-41.888
C07878=1018.523,88.784,371.081,-24.307,21.440,-41.885
C07879=1018.522,89.105,371.049,-24.307,21.439,-41.881
C07880=1018.521,89.430,371.018,-24.308,21.439,-41.879
C07881=1018.520,89.759,370.986,-24.308,21.440,-41.876
C07882=1018.519,90.092,370.954,-24.308,21.438,-41.874
C07883=1018.518,90.427,370.921,-24.309,21.439,-41.870
C07884=1018.516,90.761,370.888,-24.309,21.438,-41.866
C07885=1018.516,91.095,370.856,-24.310,21.438,-41.865
C07886=1018.515,91.430,370.823,-24.310,21.438,-41.861
C07887=1018.513,91.765,370.791,-24.311,21.438,-41.857
C07888=1018.512,92.099,370.758,-24.311,21.437,-41.855
C07889=1018.510,92.433,370.726,-24.311,21.437,-41.852
C07890=1018.510,92.768,370.694,-24.312,21.436,-41.849
C07891=1018.509,93.102,370.660,-24.312,21.437,-41.846
C07892=1018.507,93.436,370.628,-24.313,21.436,-41.842
C07893=1018.506,93.771,370.595,-24.313,21.436,-41.841
C07894=1018.505,94.106,370.562,-24.314,21.436,-41.837
C07895=1018.504,94.440,370.530,-24.314,21.436,-41.833
C07896=1018.503,94.773,370.497,-24.314,21.436,-41.832
C07897=1018.502,95.108,370.465,-24.315,21.435,-41.828
C07898=1018.500,95.442,370.432,-24.315,21.435,-41.826
C07899=1018.499,95.777,370.399,-24.316,21.435,-41.822
C07900=1018.498,96.111,370.366,-24.316,21.435,-41.819
C07901=1018.497,96.445,370.334,-24.316,21.434,-41.817
C07902=1018.496,96.779,370.302,-24.317,21.434,-41.813
C07903=1018.495,97.114,370.268,-24.317,21.434,-41.811
C07904=1018.494,97.448,370.236,-24.318,21.434,-41.808
C07905=1018.492,97.782,370.203,-24.318,21.433,-41.806
C07906=1018.491,98.116,370.170,-24.318,21.433,-41.802
C07907=1018.490,98.450,370.138,-24.319,21.433,-41.799
C07908=1018.488,98.785,370.105,-24.319,21.432,-41.796
C07909=1018.488,99.119,370.071,-24.320,21.433,-41.793
C07910=1018.486,99.454,370.039,-24.320,21.432,-41.791
C07911=1018.485,99.787,370.006,-24.320,21.432,-41.787
C07912=1018.484,100.121,369.974,-24.321,21.432,-41.785
C07913=1018.483,100.455,369.941,-24.321,21.431,-41.782
C07914=1018.481,100.789,369.908,-24.322,21.432,-41.778
C07915=1018.481,101.124,369.875,-24.322,21.431,-41.776
C07916=1018.479,101.458,369.842,-24.323,21.431,-41.773
C07917=1018.478,101.792,369.809,-24.323,21.431,-41.771
C07918=1018.477,102.126,369.776,-24.323,21.430,-41.767
C07919=1018.476,102.460,369.743,-24.324,21.430,-41.765
C07920=1018.474,102.794,369.711,-24.324,21.431,-41.762
C07921=1018.473,103.128,369.677,-24.324,21.429,-41.760
C07922=1018.472,103.463,369.644,-24.325,21.430,-41.756
C07923=1018.471,103.797,369.611,-24.325,21.429,-41.752
C07924=1018.470,104.131,369.578,-24.326,21.429,-41.751
C07925=1018.468,104.465,369.546,-24.326,21.430,-41.747
C07926=1018.467,104.799,369.512,-24.326,21.428,-41.745
C07927=1018.465,105.133,369.480,-24.327,21.429,-41.742
C07928=1018.464,105.467,369.447,-24.327,21.428,-41.739
C07929=1018.464,105.801,369.413,-24.328,21.428,-41.736
C07930=1018.462,106.135,369.380,-24.328,21.428,-41.734
C07931=1018.461,106.469,369.347,-24.328,21.427,-41.730
C07932=1018.460,106.803,369.314,-24.329,21.427,-41.728
C07933=1018.458,107.137,369.282,-24.329,21.428,-41.725
C07934=1018.457,107.471,369.248,-24.329,21.427,-41.723
C07935=1018.456,107.805,369.215,-24.330,21.427,-41.719
C07936=1018.455,108.139,369.182,-24.330,21.427,-41.718
C07937=1018.454,108.473,369.149,-24.331,21.426,-41.714
C07938=1018.453,108.807,369.116,-24.331,21.426,-41.712
C07939=1018.452,109.141,369.083,-24.332,21.426,-41.708
C07940=1018.449,109.476,369.049,-24.332,21.425,-41.706
C07941=1018.448,109.809,369.016,-24.332,21.426,-41.703
C07942=1018.447,110.143,368.983,-24.333,21.425,-41.701
C07943=1018.446,110.477,368.949,-24.333,21.425,-41.697
C07944=1018.445,110.811,368.916,-24.333,21.425,-41.695
C07945=1018.444,111.145,368.883,-24.334,21.424,-41.692
C07946=1018.443,111.479,368.851,-24.334,21.424,-41.690
C07947=1018.441,111.813,368.817,-24.335,21.425,-41.686
C07948=1018.440,112.147,368.783,-24.335,21.423,-41.684
C07949=1018.438,112.481,368.750,-24.335,21.424,-41.681
C07950=1018.438,112.815,368.717,-24.336,21.424,-41.679
C07951=1018.437,113.149,368.683,-24.336,21.423,-41.675
C07952=1018.435,113.483,368.650,-24.336,21.423,-41.673
C07953=1018.434,113.817,368.618,-24.337,21.423,-41.670
C07954=1018.432,114.151,368.584,-24.337,21.422,-41.668
C07955=1018.431,114.485,368.551,-24.338,21.423,-41.664
C07956=1018.430,114.819,368.517,-24.338,21.422,-41.662
C07957=1018.429,115.153,368.484,-24.338,21.421,-41.660
C07958=1018.428,115.486,368.451,-24.339,21.422,-41.657
C07959=1018.426,115.821,368.417,-24.339,21.422,-41.655
C07960=1018.425,116.154,368.384,-24.340,21.422,-41.652
C07961=1018.424,116.488,368.350,-24.340,21.421,-41.649
C07962=1018.423,116.822,368.317,-24.340,21.421,-41.646
C07963=1018.421,117.156,368.283,-24.341,21.421,-41.644
C07964=1018.420,117.490,368.250,-24.341,21.421,-41.640
C07965=1018.419,117.824,368.217,-24.341,21.420,-41.638
C07966=1018.418,118.158,368.183,-24.342,21.421,-41.635
C07967=1018.416,118.492,368.149,-24.342,21.420,-41.633
C07968=1018.415,118.826,368.116,-24.342,21.419,-41.631
C07969=1018.414,119.160,368.083,-24.343,21.420,-41.628
C07970=1018.412,119.494,368.049,-24.343,21.419,-41.625
C07971=1018.411,119.828,368.016,-24.344,21.419,-41.622
C07972=1018.410,120.162,367.982,-24.344,21.419,-41.620
C07973=1018.408,120.496,367.948,-24.345,21.419,-41.617
C07974=1018.407,120.830,367.915,-24.345,21.418,-41.614
C07975=1018.406,121.163,367.882,-24.345,21.418,-41.613
C07976=1018.405,121.498,367.848,-24.346,21.418,-41.609
C07977=1018.403,121.832,367.814,-24.346,21.417,-41.607
C07978=1018.403,122.165,367.781,-24.346,21.418,-41.604
C07979=1018.401,122.499,367.747,-24.347,21.418,-41.602
C07980=1018.400,122.833,367.713,-24.347,21.418,-41.598
C07981=1018.398,123.167,367.679,-24.347,21.417,-41.596
C07982=1018.397,123.501,367.646,-24.348,21.417,-41.594
C07983=1018.396,123.836,367.613,-24.348,21.417,-41.591
C07984=1018.395,124.170,367.579,-24.348,21.417,-41.589
C07985=1018.393,124.503,367.545,-24.349,21.416,-41.585
C07986=1018.392,124.837,367.511,-24.349,21.416,-41.583
C07987=1018.391,125.171,367.477,-24.349,21.416,-41.581
C07988=1018.389,125.505,367.444,-24.350,21.416,-41.578
C07989=1018.388,125.839,367.410,-24.350,21.415,-41.576
C07990=1018.387,126.174,367.376,-24.351,21.416,-41.572
C07991=1018.386,126.507,367.343,-24.351,21.415,-41.571
C07992=1018.384,126.841,367.308,-24.351,21.415,-41.569
C07993=1018.383,127.175,367.275,-24.352,21.415,-41.565
C07994=1018.381,127.509,367.241,-24.352,21.415,-41.563
C07995=1018.381,127.844,367.207,-24.352,21.414,-41.561
C07996=1018.379,128.178,367.174,-24.353,21.415,-41.558
C07997=1018.378,128.511,367.140,-24.353,21.414,-41.555
C07998=1018.377,128.846,367.105,-24.354,21.414,-41.552
C07999=1018.376,129.179,367.072,-24.354,21.414,-41.550
C08000=1018.374,129.513,367.038,-24.354,21.414,-41.548
C08001=1018.373,129.847,367.004,-24.355,21.413,-41.545
C08002=1018.371,130.181,366.970,-24.355,21.413,-41.543
C08003=1018.370,130.516,366.936,-24.355,21.413,-41.541
C08004=1018.369,130.850,366.903,-24.356,21.413,-41.538
C08005=1018.368,131.184,366.868,-24.356,21.412,-41.535
C08006=1018.367,131.518,366.835,-24.356,21.412,-41.532
C08007=1018.365,131.852,366.801,-24.357,21.412,-41.530
C08008=1018.364,132.186,366.767,-24.357,21.412,-41.528
C08009=1018.363,132.520,366.733,-24.357,21.412,-41.525
C08010=1018.361,132.854,366.699,-24.358,21.411,-41.523
C08011=1018.360,133.189,366.665,-24.358,21.411,-41.521
C08012=1018.359,133.522,366.631,-24.358,21.411,-41.517
C08013=1018.358,133.857,366.596,-24.359,21.411,-41.515
C08014=1018.356,134.191,366.563,-24.359,21.410,-41.513
C08015=1018.356,134.525,366.528,-24.359,21.411,-41.510
C08016=1018.354,134.859,366.494,-24.360,21.410,-41.508
C08017=1018.352,135.193,366.460,-24.360,21.410,-41.506
C08018=1018.352,135.526,366.426,-24.361,21.411,-41.503
C08019=1018.350,135.849,366.393,-24.361,21.410,-41.501
C08020=1018.349,136.149,366.362,-24.361,21.410,-41.499
C08021=1018.348,136.429,366.334,-24.361,21.410,-41.497
C08022=1018.347,136.694,366.307,-24.361,21.409,-41.495
C08023=1018.345,136.958,366.280,-24.362,21.409,-41.491
C08024=1018.345,137.234,366.252,-24.362,21.409,-41.490
C08025=1018.344,137.532,366.221,-24.363,21.409,-41.488
C08026=1018.342,137.854,366.189,-24.363,21.408,-41.486
C08027=1018.342,138.194,366.154,-24.363,21.408,-41.484
C08028=1018.340,138.551,366.117,-24.364,21.408,-41.480
C08029=1018.338,138.962,366.075,-24.364,21.408,-41.477
C08030=1018.337,139.190,366.052,-24.364,21.408,-41.475
C08031=1018.337,139.427,366.027,-24.365,21.408,-41.473
C08032=1018.336,139.670,366.003,-24.365,21.408,-41.473
C08033=1018.335,139.911,365.977,-24.365,21.408,-41.471
C08034=1018.333,140.143,365.954,-24.365,21.408,-41.470
C08035=1018.332,140.364,365.931,-24.365,21.407,-41.469
C08036=1018.331,140.757,365.891,-24.366,21.407,-41.465
C08037=1018.330,141.102,365.856,-24.366,21.407,-41.462
C08038=1018.328,141.441,365.820,-24.367,21.407,-41.460
C08039=1018.328,141.781,365.786,-24.367,21.407,-41.457
C08040=1018.326,142.121,365.750,-24.367,21.406,-41.455
C08041=1018.325,142.462,365.716,-24.368,21.406,-41.453
C08042=1018.324,142.803,365.680,-24.368,21.407,-41.449
C08043=1018.323,143.145,365.646,-24.368,21.406,-41.448
C08044=1018.321,143.487,365.610,-24.369,21.405,-41.445
C08045=1018.320,143.831,365.574,-24.369,21.406,-41.442
C08046=1018.319,144.174,365.540,-24.369,21.405,-41.440
C08047=1018.317,144.518,365.504,-24.370,21.405,-41.438
C08048=1018.316,144.863,365.468,-24.370,21.406,-41.435
C08049=1018.315,145.208,365.433,-24.370,21.405,-41.432
C08050=1018.314,145.553,365.397,-24.371,21.404,-41.431
C08051=1018.312,145.898,365.362,-24.371,21.405,-41.427
C08052=1018.311,146.245,365.326,-24.371,21.405,-41.425
C08053=1018.309,146.590,365.291,-24.372,21.404,-41.424
C08054=1018.302,146.937,365.259,-24.372,21.404,-41.420
C08055=1018.283,147.282,365.234,-24.372,21.404,-41.418
C08056=1018.661,147.310,364.998,-24.372,21.404,-41.418
C08057=1018.682,146.965,365.022,-24.372,21.404,-41.420
C08058=1018.690,146.618,365.053,-24.372,21.404,-41.424
C08059=1018.692,146.272,365.088,-24.371,21.405,-41.425
C08060=1018.693,145.926,365.124,-24.371,21.405,-41.427
C08061=1018.695,145.581,365.161,-24.371,21.404,-41.431
C08062=1018.696,145.235,365.196,-24.370,21.405,-41.432
C08063=1018.697,144.890,365.231,-24.370,21.406,-41.435
C08064=1018.699,144.546,365.267,-24.370,21.405,-41.438
C08065=1018.699,144.201,365.302,-24.369,21.405,-41.440
C08066=1018.701,143.859,365.338,-24.369,21.406,-41.442
C08067=1018.702,143.515,365.373,-24.369,21.405,-41.445
C08068=1018.703,143.172,365.408,-24.368,21.406,-41.448
C08069=1018.705,142.831,365.443,-24.368,21.407,-41.449
C08070=1018.706,142.489,365.479,-24.368,21.406,-41.453
C08071=1018.707,142.149,365.514,-24.367,21.406,-41.455
C08072=1018.708,141.808,365.548,-24.367,21.407,-41.457
C08073=1018.710,141.468,365.583,-24.367,21.407,-41.460
C08074=1018.711,141.130,365.618,-24.366,21.407,-41.462
C08075=1018.712,140.785,365.654,-24.366,21.407,-41.465
C08076=1018.714,140.391,365.694,-24.365,21.407,-41.469
C08077=1018.715,140.171,365.717,-24.365,21.408,-41.470
C08078=1018.715,139.937,365.740,-24.365,21.408,-41.471
C08079=1018.716,139.698,365.765,-24.365,21.408,-41.473
C08080=1018.717,139.455,365.789,-24.365,21.408,-41.473
C08081=1018.718,139.217,365.814,-24.364,21.408,-41.475
C08082=1018.719,138.990,365.838,-24.364,21.408,-41.477
C08083=1018.721,138.579,365.880,-24.364,21.408,-41.480
C08084=1018.722,138.221,365.916,-24.363,21.408,-41.484
C08085=1018.723,137.882,365.951,-24.363,21.408,-41.486
C08086=1018.725,137.559,365.984,-24.363,21.409,-41.488
C08087=1018.725,137.262,366.014,-24.362,21.409,-41.490
C08088=1018.726,136.986,366.043,-24.362,21.409,-41.491
C08089=1018.728,136.722,366.069,-24.361,21.409,-41.495
C08090=1018.729,136.457,366.097,-24.361,21.410,-41.497
C08091=1018.730,136.177,366.126,-24.361,21.410,-41.499
C08092=1018.731,135.877,366.156,-24.361,21.410,-41.501
C08093=1018.732,135.555,366.189,-24.361,21.411,-41.503
C08094=1018.734,135.221,366.223,-24.360,21.410,-41.506
C08095=1018.734,134.887,366.257,-24.360,21.410,-41.508
C08096=1018.736,134.553,366.291,-24.359,21.411,-41.510
C08097=1018.737,134.218,366.325,-24.359,21.410,-41.513
C08098=1018.738,133.884,366.359,-24.359,21.411,-41.515
C08099=1018.739,133.550,366.393,-24.358,21.411,-41.517
C08100=1018.741,133.215,366.427,-24.358,21.411,-41.521
C08101=1018.743,132.881,366.461,-24.358,21.411,-41.523
C08102=1018.743,132.548,366.496,-24.357,21.412,-41.525
C08103=1018.745,132.214,366.529,-24.357,21.412,-41.528
C08104=1018.745,131.879,366.563,-24.357,21.412,-41.530
C08105=1018.747,131.545,366.597,-24.356,21.412,-41.532
C08106=1018.748,131.211,366.632,-24.356,21.412,-41.535
C08107=1018.750,130.877,366.665,-24.356,21.413,-41.538
C08108=1018.752,130.543,366.699,-24.355,21.413,-41.541
C08109=1018.753,130.209,366.734,-24.355,21.413,-41.543
C08110=1018.754,129.875,366.767,-24.355,21.413,-41.545
C08111=1018.755,129.541,366.801,-24.354,21.414,-41.548
C08112=1018.756,129.207,366.834,-24.354,21.414,-41.550
C08113=1018.757,128.873,366.869,-24.354,21.414,-41.552
C08114=1018.758,128.539,366.902,-24.353,21.414,-41.555
C08115=1018.760,128.205,366.936,-24.353,21.415,-41.558
C08116=1018.761,127.871,366.970,-24.352,21.414,-41.561
C08117=1018.763,127.537,367.004,-24.352,21.415,-41.563
C08118=1018.763,127.203,367.038,-24.352,21.415,-41.565
C08119=1018.765,126.869,367.072,-24.351,21.415,-41.569
C08120=1018.766,126.535,367.105,-24.351,21.415,-41.571
C08121=1018.767,126.200,367.139,-24.351,21.416,-41.572
C08122=1018.769,125.867,367.172,-24.350,21.415,-41.576
C08123=1018.770,125.533,367.207,-24.350,21.416,-41.578
C08124=1018.771,125.199,367.240,-24.349,21.416,-41.581
C08125=1018.773,124.865,367.274,-24.349,21.416,-41.583
C08126=1018.774,124.531,367.307,-24.349,21.416,-41.585
C08127=1018.775,124.196,367.342,-24.348,21.417,-41.589
C08128=1018.776,123.863,367.375,-24.348,21.417,-41.591
C08129=1018.778,123.529,367.408,-24.348,21.417,-41.594
C08130=1018.779,123.195,367.443,-24.347,21.417,-41.596
C08131=1018.780,122.861,367.476,-24.347,21.418,-41.598
C08132=1018.782,122.527,367.510,-24.347,21.418,-41.602
C08133=1018.783,122.193,367.543,-24.346,21.418,-41.604
C08134=1018.783,121.859,367.577,-24.346,21.417,-41.607
C08135=1018.785,121.525,367.611,-24.346,21.418,-41.609
C08136=1018.787,121.191,367.644,-24.345,21.418,-41.613
C08137=1018.788,120.857,367.677,-24.345,21.418,-41.614
C08138=1018.789,120.523,367.711,-24.345,21.419,-41.617
C08139=1018.790,120.190,367.745,-24.344,21.419,-41.620
C08140=1018.791,119.856,367.778,-24.344,21.419,-41.622
C08141=1018.793,119.522,367.812,-24.343,21.419,-41.625
C08142=1018.794,119.187,367.846,-24.343,21.420,-41.628
C08143=1018.795,118.854,367.879,-24.342,21.419,-41.631
C08144=1018.797,118.520,367.913,-24.342,21.420,-41.633
C08145=1018.798,118.186,367.946,-24.342,21.421,-41.635
C08146=1018.799,117.852,367.979,-24.341,21.420,-41.638
C08147=1018.800,117.517,368.013,-24.341,21.421,-41.640
C08148=1018.802,117.184,368.047,-24.341,21.421,-41.644
C08149=1018.803,116.850,368.080,-24.340,21.421,-41.646
C08150=1018.804,116.516,368.113,-24.340,21.421,-41.649
C08151=1018.806,116.182,368.147,-24.340,21.422,-41.652
C08152=1018.806,115.848,368.180,-24.339,21.422,-41.655
C08153=1018.808,115.514,368.214,-24.339,21.422,-41.657
C08154=1018.809,115.180,368.247,-24.338,21.421,-41.660
C08155=1018.810,114.847,368.280,-24.338,21.422,-41.662
C08156=1018.812,114.512,368.313,-24.338,21.423,-41.664
C08157=1018.813,114.178,368.346,-24.337,21.422,-41.668
C08158=1018.814,113.844,368.380,-24.337,21.423,-41.670
C08159=1018.815,113.510,368.413,-24.336,21.423,-41.673
C08160=1018.816,113.176,368.446,-24.336,21.423,-41.675
C08161=1018.817,112.843,368.480,-24.336,21.424,-41.679
C08162=1018.819,112.509,368.514,-24.335,21.424,-41.681
C08163=1018.821,112.175,368.547,-24.335,21.423,-41.684
C08164=1018.821,111.840,368.580,-24.335,21.425,-41.686
C08165=1018.823,111.506,368.613,-24.334,21.424,-41.690
C08166=1018.824,111.172,368.646,-24.334,21.424,-41.692
C08167=1018.825,110.839,368.679,-24.333,21.425,-41.695
C08168=1018.826,110.505,368.712,-24.333,21.425,-41.697
C08169=1018.828,110.171,368.746,-24.333,21.425,-41.701
C08170=1018.829,109.836,368.779,-24.332,21.426,-41.703
C08171=1018.830,109.502,368.812,-24.332,21.425,-41.706
C08172=1018.831,109.168,368.846,-24.332,21.426,-41.708
C08173=1018.833,108.835,368.879,-24.331,21.426,-41.712
C08174=1018.834,108.501,368.912,-24.331,21.426,-41.714
C08175=1018.835,108.167,368.945,-24.330,21.427,-41.718
C08176=1018.836,107.833,368.978,-24.330,21.427,-41.719
C08177=1018.838,107.499,369.011,-24.329,21.427,-41.723
C08178=1018.838,107.164,369.044,-24.329,21.428,-41.725
C08179=1018.840,106.830,369.077,-24.329,21.427,-41.728
C08180=1018.841,106.497,369.110,-24.328,21.427,-41.730
C08181=1018.842,106.163,369.144,-24.328,21.428,-41.734
C08182=1018.843,105.829,369.176,-24.328,21.428,-41.736
C08183=1018.845,105.495,369.209,-24.327,21.428,-41.739
C08184=1018.846,105.161,369.242,-24.327,21.429,-41.742
C08185=1018.847,104.826,369.275,-24.326,21.428,-41.745
C08186=1018.848,104.492,369.309,-24.326,21.430,-41.747
C08187=1018.849,104.158,369.341,-24.326,21.429,-41.751
C08188=1018.851,103.824,369.374,-24.325,21.429,-41.752
C08189=1018.852,103.491,369.408,-24.325,21.430,-41.756
C08190=1018.853,103.156,369.440,-24.324,21.429,-41.760
C08191=1018.854,102.822,369.474,-24.324,21.431,-41.762
C08192=1018.855,102.488,369.506,-24.324,21.430,-41.765
C08193=1018.856,102.154,369.539,-24.323,21.430,-41.767
C08194=1018.858,101.819,369.572,-24.323,21.431,-41.771
C08195=1018.859,101.486,369.605,-24.323,21.431,-41.773
C08196=1018.861,101.151,369.638,-24.322,21.431,-41.776
C08197=1018.862,100.818,369.671,-24.322,21.432,-41.778
C08198=1018.863,100.483,369.704,-24.321,21.431,-41.782
C08199=1018.864,100.149,369.737,-24.321,21.432,-41.785
C08200=1018.865,99.815,369.769,-24.320,21.432,-41.787
C08201=1018.866,99.481,369.803,-24.320,21.432,-41.791
C08202=1018.868,99.147,369.835,-24.320,21.433,-41.793
C08203=1018.868,98.812,369.868,-24.319,21.432,-41.796
C08204=1018.869,98.478,369.901,-24.319,21.433,-41.799
C08205=1018.871,98.144,369.933,-24.318,21.433,-41.802
C08206=1018.872,97.810,369.966,-24.318,21.433,-41.806
C08207=1018.873,97.476,369.999,-24.318,21.434,-41.808
C08208=1018.875,97.141,370.031,-24.317,21.434,-41.811
C08209=1018.875,96.807,370.065,-24.317,21.434,-41.813
C08210=1018.877,96.473,370.097,-24.316,21.434,-41.817
C08211=1018.878,96.138,370.129,-24.316,21.435,-41.819
C08212=1018.879,95.805,370.163,-24.316,21.435,-41.822
C08213=1018.880,95.470,370.195,-24.315,21.435,-41.826
C08214=1018.881,95.135,370.228,-24.315,21.435,-41.828
C08215=1018.883,94.801,370.260,-24.314,21.436,-41.832
C08216=1018.884,94.467,370.294,-24.314,21.436,-41.833
C08217=1018.885,94.133,370.326,-24.314,21.436,-41.837
C08218=1018.886,93.798,370.358,-24.313,21.436,-41.841
C08219=1018.887,93.464,370.391,-24.313,21.436,-41.842
C08220=1018.889,93.130,370.423,-24.312,21.437,-41.846
C08221=1018.889,92.795,370.457,-24.312,21.436,-41.849
C08222=1018.891,92.461,370.490,-24.311,21.437,-41.852
C08223=1018.891,92.127,370.521,-24.311,21.437,-41.855
C08224=1018.893,91.792,370.554,-24.311,21.438,-41.857
C08225=1018.894,91.457,370.587,-24.310,21.438,-41.861
C08226=1018.895,91.123,370.619,-24.310,21.438,-41.865
C08227=1018.897,90.789,370.652,-24.309,21.438,-41.866
C08228=1018.897,90.455,370.684,-24.309,21.439,-41.870
C08229=1018.898,90.120,370.717,-24.308,21.438,-41.874
C08230=1018.899,89.787,370.749,-24.308,21.440,-41.876
C08231=1018.900,89.457,370.781,-24.308,21.439,-41.879
C08232=1018.901,89.133,370.813,-24.307,21.439,-41.881
C08233=1018.903,88.812,370.844,-24.307,21.440,-41.885
C08234=1018.903,88.491,370.875,-24.306,21.439,-41.888
C08235=1018.904,88.169,370.906,-24.306,21.441,-41.890
C08236=1018.906,87.843,370.938,-24.305,21.440,-41.894
C08237=1018.907,87.510,370.970,-24.305,21.441,-41.898
C08238=1018.908,87.173,371.003,-24.305,21.441,-41.899
C08239=1018.909,86.834,371.035,-24.304,21.441,-41.903
C08240=1018.910,86.493,371.068,-24.304,21.441,-41.906
C08241=1018.912,86.151,371.102,-24.303,21.442,-41.909
C08242=1018.913,85.808,371.135,-24.303,21.442,-41.912
C08243=1018.914,85.464,371.168,-24.302,21.442,-41.916
C08244=1018.916,85.118,371.201,-24.302,21.443,-41.918
C08245=1018.916,84.772,371.235,-24.302,21.443,-41.922
C08246=1018.918,84.424,371.269,-24.301,21.443,-41.925
C08247=1018.919,84.075,371.302,-24.301,21.443,-41.929
C08248=1018.919,83.725,371.336,-24.300,21.444,-41.931
C08249=1018.921,83.374,371.370,-24.300,21.444,-41.935
C08250=1018.921,83.022,371.404,-24.299,21.444,-41.938
C08251=1018.922,82.669,371.437,-24.299,21.444,-41.942
C08252=1018.924,82.315,371.471,-24.298,21.444,-41.945
C08253=1018.925,81.961,371.506,-24.298,21.445,-41.947
C08254=1018.927,81.605,371.540,-24.298,21.446,-41.951
C08255=1018.927,81.250,371.574,-24.297,21.445,-41.955
C08256=1018.929,80.893,371.608,-24.297,21.446,-41.958
C08257=1018.929,80.536,371.643,-24.296,21.446,-41.962
C08258=1018.931,80.182,371.677,-24.296,21.446,-41.964
C08259=1018.932,79.830,371.710,-24.295,21.447,-41.968
C08260=1018.933,79.485,371.743,-24.295,21.446,-41.971
C08261=1018.934,79.147,371.776,-24.295,21.448,-41.973
C08262=1018.935,78.814,371.808,-24.294,21.447,-41.977
C08263=1018.936,78.486,371.840,-24.293,21.448,-41.980
C08264=1018.937,78.161,371.871,-24.293,21.448,-41.984
C08265=1018.938,77.838,371.901,-24.292,21.448,-41.987
C08266=1018.938,77.514,371.933,-24.292,21.449,-41.990
C08267=1018.940,77.187,371.964,-24.292,21.449,-41.994
C08268=1018.941,76.857,371.996,-24.291,21.449,-41.997
C08269=1018.942,76.521,372.028,-24.291,21.449,-42.001
C08270=1018.943,76.179,372.060,-24.290,21.449,-42.004
C08271=1018.943,75.831,372.093,-24.290,21.450,-42.006
C08272=1018.945,75.477,372.127,-24.289,21.450,-42.010
C08273=1018.946,75.120,372.162,-24.289,21.450,-42.013
C08274=1018.947,74.762,372.195,-24.288,21.451,-42.017
C08275=1018.948,74.404,372.230,-24.288,21.451,-42.019
C08276=1018.949,74.049,372.264,-24.288,21.451,-42.023
C08277=1018.950,73.696,372.297,-24.287,21.452,-42.027
C08278=1018.951,73.344,372.331,-24.286,21.451,-42.030
C08279=1018.953,72.995,372.364,-24.286,21.452,-42.034
C08280=1018.954,72.647,372.396,-24.285,21.452,-42.037
C08281=1018.955,72.301,372.430,-24.285,21.453,-42.041
C08282=1018.955,71.955,372.463,-24.285,21.453,-42.043
C08283=1018.957,71.610,372.495,-24.284,21.453,-42.047
C08284=1018.957,71.266,372.528,-24.284,21.454,-42.051
C08285=1018.959,70.922,372.560,-24.283,21.453,-42.054
C08286=1018.960,70.577,372.593,-24.283,21.454,-42.058
C08287=1018.960,70.232,372.626,-24.282,21.454,-42.061
C08288=1018.962,69.888,372.659,-24.282,21.455,-42.063
C08289=1018.963,69.544,372.691,-24.281,21.455,-42.067
C08290=1018.963,69.201,372.724,-24.281,21.456,-42.071
C08291=1018.964,68.859,372.756,-24.280,21.455,-42.074
C08292=1018.965,68.517,372.789,-24.280,21.456,-42.078
C08293=1018.966,68.177,372.821,-24.279,21.456,-42.082
C08294=1018.967,67.838,372.853,-24.279,21.456,-42.085
C08295=1018.969,67.499,372.885,-24.279,21.457,-42.087
C08296=1018.969,67.162,372.917,-24.278,21.457,-42.091
C08297=1018.970,66.825,372.949,-24.278,21.457,-42.094
C08298=1018.971,66.490,372.980,-24.277,21.457,-42.098
C08299=1018.972,66.157,373.012,-24.277,21.458,-42.102
C08300=1018.974,65.818,373.044,-24.276,21.457,-42.105
C08301=1018.974,65.464,373.077,-24.276,21.459,-42.108
C08302=1018.975,65.087,373.113,-24.275,21.458,-42.113
C08303=1018.977,64.691,373.150,-24.274,21.459,-42.116
C08304=1018.977,64.305,373.186,-24.274,21.459,-42.120
C08305=1018.978,63.949,373.219,-24.274,21.460,-42.124
C08306=1018.979,63.575,373.255,-24.273,21.460,-42.128
C08307=1018.980,63.356,373.276,-24.273,21.461,-42.130
C08308=1018.983,63.133,373.295,-24.272,21.460,-42.131
C08309=1018.988,62.737,373.330,-24.272,21.460,-42.135
C08310=1018.992,62.400,373.359,-24.271,21.461,-42.139
C08311=1018.996,62.065,373.389,-24.271,21.461,-42.142
C08312=1019.001,61.730,373.417,-24.270,21.462,-42.146
C08313=1019.004,61.396,373.447,-24.270,21.461,-42.149
C08314=1019.009,61.060,373.477,-24.269,21.462,-42.153
C08315=1019.013,60.725,373.506,-24.269,21.462,-42.157
C08316=1019.017,60.391,373.536,-24.268,21.462,-42.160
C08317=1019.022,60.055,373.565,-24.268,21.463,-42.163
C08318=1019.025,59.720,373.595,-24.268,21.464,-42.166
C08319=1019.029,59.385,373.624,-24.267,21.464,-42.170
C08320=1019.033,59.050,373.653,-24.267,21.464,-42.173
C08321=1019.038,58.715,373.682,-24.266,21.464,-42.177
C08322=1019.042,58.380,373.712,-24.266,21.465,-42.181
C08323=1019.045,58.045,373.741,-24.265,21.464,-42.184
C08324=1019.049,57.710,373.770,-24.264,21.465,-42.188
C08325=1019.053,57.375,373.799,-24.264,21.465,-42.192
C08326=1019.057,57.041,373.829,-24.264,21.466,-42.194
C08327=1019.062,56.705,373.858,-24.263,21.466,-42.197
C08328=1019.065,56.370,373.888,-24.263,21.466,-42.201
C08329=1019.069,56.035,373.917,-24.262,21.467,-42.205
C08330=1019.073,55.700,373.946,-24.262,21.467,-42.209
C08331=1019.077,55.364,373.975,-24.261,21.467,-42.212
C08332=1019.081,55.030,374.004,-24.261,21.467,-42.216
C08333=1019.085,54.695,374.033,-24.260,21.468,-42.220
C08334=1019.089,54.360,374.063,-24.260,21.468,-42.223
C08335=1019.093,54.025,374.092,-24.259,21.468,-42.227
C08336=1019.096,53.690,374.122,-24.259,21.468,-42.230
C08337=1019.100,53.355,374.151,-24.258,21.469,-42.234
C08338=1019.104,53.020,374.180,-24.258,21.469,-42.238
C08339=1019.108,52.685,374.209,-24.257,21.470,-42.240
C08340=1019.112,52.350,374.238,-24.257,21.470,-42.244
C08341=1019.115,52.015,374.268,-24.256,21.470,-42.247
C08342=1019.119,51.680,374.297,-24.256,21.471,-42.251
C08343=1019.123,51.345,374.326,-24.255,21.471,-42.254
C08344=1019.126,51.010,374.355,-24.255,21.471,-42.258
C08345=1019.130,50.674,374.384,-24.254,21.471,-42.262
C08346=1019.134,50.340,374.413,-24.254,21.472,-42.266
C08347=1019.137,50.004,374.442,-24.253,21.472,-42.269
C08348=1019.142,49.670,374.471,-24.253,21.472,-42.273
C08349=1019.146,49.335,374.500,-24.252,21.473,-42.277
C08350=1019.148,49.000,374.529,-24.252,21.473,-42.280
C08351=1019.152,48.665,374.558,-24.251,21.473,-42.284
C08352=1019.156,48.330,374.588,-24.251,21.473,-42.287
C08353=1019.159,47.995,374.616,-24.250,21.474,-42.291
C08354=1019.163,47.660,374.646,-24.250,21.474,-42.295
C08355=1019.167,47.325,374.675,-24.249,21.475,-42.299
C08356=1019.170,46.990,374.704,-24.249,21.475,-42.302
C08357=1019.173,46.655,374.733,-24.248,21.475,-42.306
C08358=1019.177,46.320,374.762,-24.248,21.475,-42.309
C08359=1019.181,45.985,374.790,-24.247,21.476,-42.313
C08360=1019.184,45.651,374.820,-24.247,21.476,-42.317
C08361=1019.188,45.315,374.849,-24.246,21.477,-42.321
C08362=1019.191,44.981,374.878,-24.246,21.477,-42.325
C08363=1019.195,44.645,374.907,-24.245,21.477,-42.328
C08364=1019.198,44.311,374.936,-24.245,21.477,-42.332
C08365=1019.202,43.975,374.965,-24.244,21.478,-42.335
C08366=1019.205,43.641,374.994,-24.244,21.478,-42.339
C08367=1019.209,43.305,375.023,-24.243,21.479,-42.343
C08368=1019.212,42.971,375.052,-24.243,21.479,-42.347
C08369=1019.216,42.635,375.081,-24.242,21.479,-42.350
C08370=1019.219,42.302,375.109,-24.242,21.479,-42.354
C08371=1019.222,41.967,375.138,-24.241,21.480,-42.357
C08372=1019.226,41.632,375.167,-24.241,21.480,-42.361
C08373=1019.229,41.297,375.196,-24.240,21.481,-42.365
C08374=1019.233,40.962,375.225,-24.240,21.481,-42.369
C08375=1019.235,40.627,375.254,-24.239,21.481,-42.372
C08376=1019.239,40.292,375.282,-24.239,21.481,-42.376
C08377=1019.242,39.957,375.312,-24.238,21.482,-42.380
C08378=1019.245,39.622,375.340,-24.238,21.482,-42.383
C08379=1019.248,39.288,375.369,-24.237,21.483,-42.387
C08380=1019.251,38.953,375.398,-24.237,21.483,-42.391
C08381=1019.256,38.619,375.427,-24.236,21.483,-42.395
C08382=1019.259,38.284,375.455,-24.236,21.483,-42.398
C08383=1019.262,37.949,375.484,-24.235,21.484,-42.402
C08384=1019.265,37.614,375.513,-24.235,21.484,-42.405
C08385=1019.268,37.279,375.542,-24.234,21.485,-42.409
C08386=1019.271,36.944,375.570,-24.234,21.485,-42.413
C08387=1019.274,36.610,375.599,-24.233,21.485,-42.418
C08388=1019.277,36.275,375.629,-24.232,21.485,-42.422
C08389=1019.281,35.941,375.657,-24.232,21.486,-42.426
C08390=1019.284,35.606,375.686,-24.231,21.485,-42.429
C08391=1019.287,35.271,375.714,-24.231,21.486,-42.433
C08392=1019.290,34.937,375.743,-24.230,21.486,-42.437
C08393=1019.293,34.601,375.771,-24.230,21.487,-42.440
C08394=1019.296,34.267,375.800,-24.229,21.487,-42.444
C08395=1019.299,33.932,375.829,-24.229,21.488,-42.448
C08396=1019.303,33.598,375.857,-24.228,21.488,-42.452
C08397=1019.305,33.264,375.886,-24.228,21.489,-42.455
C08398=1019.308,32.929,375.914,-24.227,21.489,-42.459
C08399=1019.311,32.594,375.943,-24.226,21.489,-42.464
C08400=1019.314,32.259,375.971,-24.226,21.489,-42.468
C08401=1019.317,31.925,376.000,-24.225,21.489,-42.471
C08402=1019.321,31.590,376.028,-24.225,21.490,-42.475
C08403=1019.323,31.256,376.057,-24.224,21.490,-42.479
C08404=1019.326,30.922,376.086,-24.224,21.491,-42.483
C08405=1019.329,30.586,376.114,-24.223,21.491,-42.486
C08406=1019.332,30.252,376.143,-24.223,21.492,-42.490
C08407=1019.335,29.918,376.171,-24.222,21.492,-42.494
C08408=1019.338,29.583,376.200,-24.222,21.493,-42.498
C08409=1019.341,29.249,376.229,-24.221,21.492,-42.503
C08410=1019.343,28.914,376.256,-24.221,21.493,-42.507
C08411=1019.346,28.580,376.285,-24.220,21.493,-42.510
C08412=1019.349,28.246,376.314,-24.220,21.494,-42.514
C08413=1019.352,27.911,376.342,-24.219,21.494,-42.518
C08414=1019.355,27.577,376.371,-24.219,21.495,-42.522
C08415=1019.357,27.242,376.399,-24.218,21.494,-42.525
C08416=1019.360,26.908,376.427,-24.217,21.494,-42.530
C08417=1019.363,26.574,376.456,-24.217,21.495,-42.534
C08418=1019.365,26.239,376.485,-24.216,21.495,-42.538
C08419=1019.369,25.905,376.512,-24.216,21.496,-42.541
C08420=1019.371,25.571,376.541,-24.215,21.496,-42.545
C08421=1019.374,25.237,376.569,-24.215,21.497,-42.549
C08422=1019.377,24.901,376.598,-24.214,21.497,-42.553
C08423=1019.379,24.568,376.626,-24.213,21.497,-42.558
C08424=1019.382,24.242,376.653,-24.213,21.498,-42.560
C08425=1019.384,23.946,376.678,-24.213,21.498,-42.562
C08426=1019.386,23.694,376.700,-24.212,21.498,-42.565
C08427=1019.389,23.286,376.734,-24.211,21.499,-42.573
C08428=1019.393,22.877,376.769,-24.210,21.499,-42.580
C08429=1019.395,22.624,376.790,-24.210,21.500,-42.582
C08430=1019.397,22.330,376.815,-24.210,21.501,-42.584
C08431=1019.399,22.006,376.842,-24.209,21.500,-42.588
C08432=1019.402,21.649,376.872,-24.209,21.501,-42.593
C08433=1019.404,21.442,376.890,-24.208,21.501,-42.597
C08434=1019.406,21.215,376.910,-24.208,21.502,-42.599
C08435=1019.407,20.973,376.929,-24.208,21.502,-42.601
C08436=1019.409,20.725,376.951,-24.207,21.502,-42.603
C08437=1019.411,20.479,376.971,-24.207,21.502,-42.604
C08438=1019.413,20.242,376.991,-24.207,21.502,-42.608
C08439=1019.416,19.825,377.026,-24.206,21.503,-42.613
C08440=1019.418,19.477,377.056,-24.205,21.502,-42.619
C08441=1019.421,19.145,377.084,-24.205,21.503,-42.622
C08442=1019.424,18.813,377.112,-24.204,21.503,-42.626
C08443=1019.426,18.481,377.140,-24.204,21.504,-42.630
C08444=1019.428,18.150,377.167,-24.203,21.504,-42.634
C08445=1019.431,17.820,377.195,-24.202,21.504,-42.639
C08446=1019.433,17.490,377.222,-24.202,21.505,-42.643
C08447=1019.436,17.161,377.251,-24.201,21.505,-42.646
C08448=1019.438,16.832,377.278,-24.201,21.506,-42.650
C08449=1019.440,16.505,377.305,-24.200,21.506,-42.654
C08450=1019.443,16.177,377.333,-24.200,21.507,-42.658
C08451=1019.445,15.850,377.360,-24.199,21.507,-42.663
C08452=1019.447,15.524,377.388,-24.199,21.507,-42.667
C08453=1019.450,15.197,377.415,-24.198,21.508,-42.670
C08454=1019.451,14.872,377.442,-24.198,21.508,-42.674
C08455=1019.454,14.547,377.470,-24.197,21.509,-42.678
C08456=1019.456,14.223,377.497,-24.197,21.509,-42.682
C08457=1019.458,13.898,377.523,-24.196,21.509,-42.687
C08458=1019.461,13.573,377.551,-24.195,21.509,-42.691
C08459=1019.463,13.250,377.579,-24.195,21.510,-42.694
C08460=1019.465,12.926,377.605,-24.194,21.510,-42.698
C08461=1019.467,12.603,377.632,-24.194,21.511,-42.702
C08462=1019.469,12.279,377.659,-24.193,21.511,-42.707
C08463=1019.471,11.955,377.686,-24.193,21.511,-42.711
C08464=1019.473,11.633,377.713,-24.192,21.512,-42.715
C08465=1019.476,11.310,377.740,-24.192,21.512,-42.718
C08466=1019.477,10.990,377.767,-24.191,21.513,-42.722
C08467=1019.480,10.671,377.793,-24.191,21.513,-42.726
C08468=1019.482,10.354,377.819,-24.190,21.514,-42.730
C08469=1019.484,10.039,377.846,-24.190,21.514,-42.733
C08470=1019.486,9.723,377.872,-24.189,21.514,-42.738
C08471=1019.488,9.409,377.898,-24.188,21.515,-42.742
C08472=1019.490,9.093,377.924,-24.188,21.515,-42.746
C08473=1019.492,8.777,377.951,-24.187,21.516,-42.750
C08474=1019.494,8.458,377.977,-24.186,21.515,-42.755
C08475=1019.495,8.138,378.004,-24.186,21.516,-42.759
C08476=1019.498,7.815,378.031,-24.186,21.516,-42.762
C08477=1019.499,7.489,378.058,-24.185,21.517,-42.766
C08478=1019.501,7.161,378.085,-24.185,21.517,-42.770
C08479=1019.503,6.834,378.112,-24.184,21.518,-42.774
C08480=1019.506,6.505,378.140,-24.183,21.518,-42.779
C08481=1019.507,6.175,378.167,-24.183,21.518,-42.783
C08482=1019.509,5.846,378.194,-24.182,21.519,-42.786
C08483=1019.511,5.515,378.221,-24.181,21.518,-42.792
C08484=1019.513,5.185,378.248,-24.181,21.519,-42.795
C08485=1019.515,4.853,378.276,-24.180,21.519,-42.799
C08486=1019.517,4.521,378.303,-24.180,21.521,-42.803
C08487=1019.519,4.192,378.331,-24.179,21.520,-42.807
C08488=1019.520,3.878,378.356,-24.179,21.521,-42.810
C08489=1019.522,3.590,378.380,-24.179,21.521,-42.814
C08490=1019.524,3.319,378.403,-24.178,21.522,-42.818
C08491=1019.525,3.058,378.424,-24.177,21.522,-42.823
C08492=1019.526,2.789,378.446,-24.177,21.522,-42.827
C08493=1019.529,2.501,378.470,-24.176,21.523,-42.831
C08494=1019.530,2.189,378.496,-24.176,21.523,-42.834
C08495=1019.532,1.858,378.523,-24.175,21.523,-42.838
C08496=1019.534,1.524,378.551,-24.175,21.524,-42.842
C08497=1019.536,1.191,378.578,-24.174,21.525,-42.846
C08498=1019.537,0.856,378.606,-24.173,21.525,-42.851
C08499=1019.539,0.520,378.633,-24.173,21.525,-42.855
C08500=1019.540,0.183,378.661,-24.172,21.526,-42.858
C08501=1019.542,-0.156,378.689,-24.172,21.526,-42.864
C08502=1019.544,-0.496,378.716,-24.171,21.526,-42.867
C08503=1019.546,-0.838,378.745,-24.170,21.527,-42.873
C08504=1019.548,-1.182,378.773,-24.170,21.527,-42.877
C08505=1019.550,-1.526,378.801,-24.169,21.528,-42.880
C08506=1019.551,-1.873,378.830,-24.169,21.528,-42.886
C08507=1019.553,-2.221,378.858,-24.168,21.529,-42.890
C08508=1019.555,-2.571,378.886,-24.167,21.529,-42.895
C08509=1019.557,-2.923,378.916,-24.167,21.529,-42.899
C08510=1019.558,-3.274,378.944,-24.166,21.529,-42.904
C08511=1019.560,-3.629,378.974,-24.166,21.531,-42.908
C08512=1019.561,-3.986,379.002,-24.165,21.530,-42.913
C08513=1019.563,-4.348,379.032,-24.164,21.531,-42.919
C08514=1019.565,-4.714,379.062,-24.164,21.532,-42.923
C08515=1019.566,-5.085,379.092,-24.163,21.532,-42.928
C08516=1019.568,-5.459,379.122,-24.163,21.533,-42.932
C08517=1019.570,-5.834,379.153,-24.162,21.533,-42.937
C08518=1019.571,-6.209,379.184,-24.161,21.533,-42.941
C08519=1019.574,-6.584,379.214,-24.160,21.534,-42.947
C08520=1019.575,-6.956,379.245,-24.160,21.534,-42.952
C08521=1019.576,-7.325,379.274,-24.159,21.535,-42.956
C08522=1019.578,-7.690,379.305,-24.158,21.535,-42.961
C08523=1019.580,-8.054,379.334,-24.158,21.536,-42.967
C08524=1019.581,-8.417,379.363,-24.157,21.536,-42.971
C08525=1019.583,-8.780,379.393,-24.156,21.536,-42.976
C08526=1019.585,-9.142,379.422,-24.156,21.537,-42.982
C08527=1019.586,-9.505,379.452,-24.155,21.538,-42.985
C08528=1019.587,-9.866,379.481,-24.154,21.538,-42.991
C08529=1019.589,-10.227,379.511,-24.154,21.539,-42.995
C08530=1019.590,-10.587,379.540,-24.153,21.539,-43.000
C08531=1019.591,-10.946,379.568,-24.152,21.539,-43.006
C08532=1019.593,-11.303,379.598,-24.152,21.540,-43.009
C08533=1019.594,-11.660,379.626,-24.151,21.540,-43.014
C08534=1019.596,-12.015,379.654,-24.151,21.541,-43.019
C08535=1019.597,-12.368,379.684,-24.150,21.541,-43.024
C08536=1019.599,-12.720,379.712,-24.149,21.542,-43.028
C08537=1019.599,-13.070,379.740,-24.149,21.542,-43.033
C08538=1019.601,-13.419,379.768,-24.148,21.543,-43.037
C08539=1019.602,-13.766,379.796,-24.147,21.543,-43.042
C08540=1019.603,-14.109,379.824,-24.147,21.544,-43.046
C08541=1019.605,-14.452,379.851,-24.146,21.544,-43.052
C08542=1019.606,-14.792,379.879,-24.146,21.544,-43.055
C08543=1019.608,-15.130,379.906,-24.145,21.545,-43.061
C08544=1019.608,-15.466,379.933,-24.145,21.546,-43.065
C08545=1019.609,-15.801,379.960,-24.144,21.546,-43.070
C08546=1019.610,-16.136,379.987,-24.143,21.546,-43.074
C08547=1019.611,-16.470,380.014,-24.142,21.547,-43.079
C08548=1019.613,-16.803,380.041,-24.142,21.547,-43.083
C08549=1019.614,-17.135,380.068,-24.141,21.547,-43.088
C08550=1019.615,-17.469,380.093,-24.141,21.548,-43.092
C08551=1019.616,-17.834,380.123,-24.140,21.549,-43.100
C08552=1019.617,-18.056,380.140,-24.139,21.548,-43.103
C08553=1019.617,-18.303,380.160,-24.139,21.549,-43.105
C08554=1019.618,-18.564,380.182,-24.139,21.550,-43.107
C08555=1019.619,-18.826,380.203,-24.139,21.550,-43.109
C08556=1019.619,-19.073,380.222,-24.138,21.550,-43.112
C08557=1019.621,-19.491,380.255,-24.137,21.550,-43.118
C08558=1019.621,-19.663,380.270,-24.137,21.551,-43.122
C08559=1019.622,-19.996,380.296,-24.136,21.551,-43.127
C08560=1019.623,-20.329,380.323,-24.136,21.552,-43.131
C08561=1019.624,-20.661,380.349,-24.135,21.553,-43.135
C08562=1019.625,-20.994,380.376,-24.134,21.552,-43.140
C08563=1019.625,-21.327,380.402,-24.134,21.553,-43.144
C08564=1019.627,-21.660,380.428,-24.133,21.554,-43.149
C08565=1019.627,-21.993,380.455,-24.133,21.554,-43.153
C08566=1019.629,-22.325,380.482,-24.132,21.554,-43.158
C08567=1019.629,-22.658,380.508,-24.131,21.556,-43.162
C08568=1019.630,-22.991,380.535,-24.131,21.555,-43.168
C08569=1019.631,-23.323,380.561,-24.130,21.556,-43.171
C08570=1019.632,-23.656,380.588,-24.129,21.556,-43.177
C08571=1019.633,-23.989,380.613,-24.129,21.557,-43.181
C08572=1019.634,-24.322,380.640,-24.128,21.557,-43.186
C08573=1019.634,-24.655,380.667,-24.128,21.558,-43.190
C08574=1019.635,-24.988,380.693,-24.127,21.558,-43.195
C08575=1019.635,-25.320,380.720,-24.126,21.559,-43.199
C08576=1019.637,-25.654,380.746,-24.126,21.559,-43.204
C08577=1019.637,-25.986,380.772,-24.125,21.559,-43.208
C08578=1019.638,-26.319,380.798,-24.124,21.560,-43.214
C08579=1019.638,-26.651,380.825,-24.124,21.560,-43.217
C08580=1019.640,-26.984,380.851,-24.123,21.560,-43.223
C08581=1019.640,-27.317,380.877,-24.123,21.562,-43.227
C08582=1019.641,-27.650,380.903,-24.122,21.562,-43.232
C08583=1019.641,-27.982,380.930,-24.121,21.562,-43.236
C08584=1019.642,-28.315,380.956,-24.120,21.562,-43.241
C08585=1019.643,-28.648,380.983,-24.120,21.563,-43.245
C08586=1019.643,-28.982,381.009,-24.119,21.563,-43.250
C08587=1019.644,-29.314,381.035,-24.119,21.564,-43.254
C08588=1019.644,-29.647,381.061,-24.118,21.565,-43.260
C08589=1019.645,-29.979,381.088,-24.118,21.565,-43.264
C08590=1019.646,-30.312,381.113,-24.117,21.565,-43.269
C08591=1019.646,-30.645,381.139,-24.116,21.566,-43.273
C08592=1019.647,-30.977,381.166,-24.116,21.566,-43.278
C08593=1019.647,-31.310,381.192,-24.115,21.567,-43.282
C08594=1019.648,-31.643,381.218,-24.114,21.567,-43.287
C08595=1019.649,-31.975,381.244,-24.114,21.568,-43.291
C08596=1019.648,-32.309,381.270,-24.113,21.568,-43.296
C08597=1019.649,-32.641,381.297,-24.113,21.569,-43.301
C08598=1019.649,-32.974,381.322,-24.112,21.569,-43.306
C08599=1019.650,-33.307,381.348,-24.111,21.570,-43.310
C08600=1019.650,-33.639,381.374,-24.111,21.570,-43.315
C08601=1019.651,-33.972,381.400,-24.110,21.571,-43.319
C08602=1019.651,-34.305,381.426,-24.109,21.571,-43.324
C08603=1019.652,-34.637,381.452,-24.109,21.572,-43.328
C08604=1019.652,-34.969,381.478,-24.108,21.572,-43.334
C08605=1019.652,-35.303,381.504,-24.108,21.573,-43.337
C08606=1019.653,-35.635,381.530,-24.107,21.573,-43.343
C08607=1019.652,-35.968,381.556,-24.107,21.574,-43.347
C08608=1019.653,-36.301,381.582,-24.106,21.574,-43.352
C08609=1019.653,-36.634,381.608,-24.105,21.574,-43.357
C08610=1019.653,-36.966,381.634,-24.105,21.575,-43.361
C08611=1019.654,-37.299,381.659,-24.104,21.575,-43.366
C08612=1019.655,-37.632,381.685,-24.103,21.576,-43.371
C08613=1019.654,-37.964,381.711,-24.102,21.576,-43.376
C08614=1019.655,-38.297,381.737,-24.102,21.577,-43.380
C08615=1019.655,-38.629,381.762,-24.101,21.577,-43.385
C08616=1019.655,-38.962,381.789,-24.101,21.578,-43.389
C08617=1019.656,-39.294,381.814,-24.100,21.578,-43.394
C08618=1019.655,-39.628,381.840,-24.100,21.579,-43.398
C08619=1019.655,-39.960,381.866,-24.099,21.579,-43.404
C08620=1019.656,-40.293,381.892,-24.098,21.580,-43.409
C08621=1019.656,-40.625,381.917,-24.098,21.580,-43.413
C08622=1019.656,-40.958,381.944,-24.097,21.580,-43.418
C08623=1019.656,-41.290,381.968,-24.096,21.582,-43.422
C08624=1019.656,-41.623,381.994,-24.096,21.582,-43.427
C08625=1019.657,-41.955,382.020,-24.095,21.582,-43.431
C08626=1019.657,-42.288,382.045,-24.094,21.583,-43.437
C08627=1019.657,-42.620,382.071,-24.094,21.583,-43.442
C08628=1019.657,-42.953,382.097,-24.093,21.583,-43.446
C08629=1019.657,-43.286,382.122,-24.092,21.584,-43.451
C08630=1019.656,-43.618,382.148,-24.092,21.585,-43.455
C08631=1019.656,-43.951,382.173,-24.091,21.585,-43.461
C08632=1019.657,-44.284,382.200,-24.091,21.586,-43.465
C08633=1019.657,-44.616,382.225,-24.090,21.586,-43.470
C08634=1019.657,-44.949,382.250,-24.089,21.586,-43.475
C08635=1019.656,-45.281,382.276,-24.089,21.587,-43.479
C08636=1019.657,-45.614,382.301,-24.088,21.588,-43.485
C08637=1019.656,-45.946,382.327,-24.088,21.588,-43.488
C08638=1019.656,-46.278,382.352,-24.087,21.588,-43.494
C08639=1019.656,-46.611,382.377,-24.086,21.590,-43.498
C08640=1019.656,-46.943,382.403,-24.086,21.589,-43.503
C08641=1019.656,-47.276,382.429,-24.085,21.589,-43.508
C08642=1019.657,-47.609,382.454,-24.084,21.591,-43.512
C08643=1019.656,-47.941,382.479,-24.083,21.591,-43.518
C08644=1019.656,-48.273,382.504,-24.083,21.592,-43.522
C08645=1019.655,-48.606,382.530,-24.082,21.592,-43.527
C08646=1019.655,-48.938,382.556,-24.081,21.592,-43.532
C08647=1019.655,-49.271,382.581,-24.081,21.593,-43.536
C08648=1019.654,-49.603,382.607,-24.080,21.593,-43.542
C08649=1019.655,-49.936,382.632,-24.080,21.595,-43.546
C08650=1019.654,-50.269,382.657,-24.079,21.594,-43.551
C08651=1019.653,-50.600,382.683,-24.079,21.595,-43.555
C08652=1019.653,-50.933,382.708,-24.078,21.596,-43.560
C08653=1019.653,-51.265,382.733,-24.077,21.596,-43.566
C08654=1019.654,-51.598,382.758,-24.077,21.597,-43.570
C08655=1019.653,-51.929,382.783,-24.076,21.597,-43.575
C08656=1019.653,-52.262,382.809,-24.075,21.597,-43.579
C08657=1019.653,-52.594,382.834,-24.075,21.598,-43.584
C08658=1019.652,-52.926,382.859,-24.074,21.598,-43.589
C08659=1019.652,-53.259,382.884,-24.074,21.600,-43.594
C08660=1019.652,-53.591,382.909,-24.073,21.599,-43.599
C08661=1019.651,-53.923,382.934,-24.072,21.600,-43.603
C08662=1019.651,-54.256,382.959,-24.072,21.601,-43.608
C08663=1019.650,-54.588,382.984,-24.071,21.601,-43.613
C08664=1019.650,-54.921,383.009,-24.070,21.602,-43.618
C08665=1019.649,-55.253,383.035,-24.070,21.602,-43.623
C08666=1019.648,-55.586,383.060,-24.069,21.603,-43.627
C08667=1019.648,-55.919,383.085,-24.068,21.603,-43.632
C08668=1019.647,-56.251,383.110,-24.068,21.603,-43.637
C08669=1019.647,-56.584,383.135,-24.067,21.605,-43.642
C08670=1019.646,-56.918,383.161,-24.066,21.604,-43.647
C08671=1019.646,-57.252,383.185,-24.066,21.605,-43.652
C08672=1019.646,-57.586,383.211,-24.065,21.606,-43.656
C08673=1019.645,-57.920,383.235,-24.064,21.606,-43.662
C08674=1019.644,-58.254,383.261,-24.064,21.607,-43.666
C08675=1019.644,-58.589,383.286,-24.063,21.607,-43.671
C08676=1019.643,-58.924,383.310,-24.062,21.608,-43.676
C08677=1019.642,-59.260,383.336,-24.062,21.608,-43.680
C08678=1019.642,-59.597,383.361,-24.061,21.609,-43.686
C08679=1019.641,-59.933,383.387,-24.060,21.609,-43.691
C08680=1019.641,-60.270,383.411,-24.060,21.610,-43.695
C08681=1019.640,-60.607,383.437,-24.059,21.610,-43.700
C08682=1019.639,-60.945,383.462,-24.059,21.611,-43.706
C08683=1019.638,-61.282,383.487,-24.058,21.611,-43.710
C08684=1019.637,-61.621,383.513,-24.057,21.612,-43.715
C08685=1019.636,-61.960,383.538,-24.057,21.612,-43.720
C08686=1019.636,-62.299,383.564,-24.056,21.614,-43.725
C08687=1019.636,-62.639,383.589,-24.055,21.613,-43.730
C08688=1019.634,-62.978,383.614,-24.055,21.614,-43.735
C08689=1019.633,-63.319,383.639,-24.054,21.615,-43.739
C08690=1019.633,-63.659,383.665,-24.053,21.616,-43.745
C08691=1019.632,-64.000,383.689,-24.053,21.615,-43.750
C08692=1019.632,-64.342,383.715,-24.052,21.617,-43.754
C08693=1019.631,-64.683,383.740,-24.051,21.617,-43.759
C08694=1019.630,-65.025,383.766,-24.051,21.618,-43.765
C08695=1019.629,-65.367,383.792,-24.050,21.617,-43.770
C08696=1019.627,-65.709,383.817,-24.050,21.619,-43.774
C08697=1019.627,-66.052,383.842,-24.049,21.619,-43.780
C08698=1019.625,-66.395,383.868,-24.048,21.620,-43.785
C08699=1019.624,-66.738,383.893,-24.048,21.620,-43.789
C08700=1019.624,-67.081,383.919,-24.047,21.621,-43.795
C08701=1019.623,-67.424,383.944,-24.046,21.621,-43.800
C08702=1019.622,-67.767,383.969,-24.045,21.622,-43.805
C08703=1019.621,-68.111,383.994,-24.045,21.622,-43.809
C08704=1019.620,-68.454,384.020,-24.044,21.623,-43.815
C08705=1019.619,-68.799,384.045,-24.043,21.623,-43.820
C08706=1019.618,-69.143,384.071,-24.043,21.624,-43.824
C08707=1019.616,-69.487,384.096,-24.042,21.624,-43.829
C08708=1019.615,-69.830,384.121,-24.041,21.625,-43.835
C08709=1019.614,-70.174,384.146,-24.041,21.625,-43.840
C08710=1019.613,-70.519,384.171,-24.040,21.626,-43.844
C08711=1019.612,-70.863,384.197,-24.040,21.627,-43.850
C08712=1019.611,-71.207,384.222,-24.039,21.627,-43.855
C08713=1019.610,-71.551,384.248,-24.038,21.628,-43.861
C08714=1019.608,-71.894,384.273,-24.038,21.628,-43.865
C08715=1019.607,-72.239,384.298,-24.037,21.629,-43.870
C08716=1019.606,-72.583,384.324,-24.036,21.629,-43.875
C08717=1019.604,-72.927,384.348,-24.035,21.630,-43.881
C08718=1019.604,-73.270,384.373,-24.035,21.630,-43.885
C08719=1019.602,-73.614,384.399,-24.034,21.631,-43.890
C08720=1019.601,-73.958,384.424,-24.033,21.632,-43.896
C08721=1019.599,-74.301,384.448,-24.033,21.632,-43.901
C08722=1019.598,-74.645,384.474,-24.032,21.633,-43.905
C08723=1019.597,-74.988,384.499,-24.031,21.633,-43.911
C08724=1019.595,-75.331,384.524,-24.031,21.634,-43.916
C08725=1019.595,-75.674,384.549,-24.030,21.634,-43.920
C08726=1019.593,-76.017,384.574,-24.030,21.635,-43.926
C08727=1019.592,-76.360,384.599,-24.029,21.635,-43.931
C08728=1019.590,-76.703,384.624,-24.028,21.636,-43.936
C08729=1019.588,-77.045,384.649,-24.028,21.636,-43.940
C08730=1019.587,-77.387,384.674,-24.027,21.637,-43.946
C08731=1019.586,-77.728,384.699,-24.026,21.637,-43.951
C08732=1019.584,-78.070,384.723,-24.026,21.639,-43.955
C08733=1019.582,-78.411,384.748,-24.025,21.638,-43.960
C08734=1019.582,-78.752,384.773,-24.024,21.639,-43.966
C08735=1019.580,-79.093,384.797,-24.023,21.639,-43.971
C08736=1019.578,-79.433,384.822,-24.023,21.641,-43.975
C08737=1019.577,-79.772,384.846,-24.022,21.641,-43.981
C08738=1019.575,-80.112,384.871,-24.021,21.641,-43.986
C08739=1019.574,-80.451,384.895,-24.021,21.643,-43.990
C08740=1019.572,-80.789,384.920,-24.020,21.643,-43.995
C08741=1019.571,-81.128,384.944,-24.020,21.643,-44.001
C08742=1019.569,-81.466,384.969,-24.019,21.644,-44.005
C08743=1019.567,-81.803,384.994,-24.018,21.645,-44.010
C08744=1019.565,-82.140,385.017,-24.018,21.645,-44.016
C08745=1019.564,-82.476,385.042,-24.017,21.645,-44.021
C08746=1019.562,-82.812,385.066,-24.016,21.646,-44.025
C08747=1019.561,-83.148,385.090,-24.016,21.647,-44.031
C08748=1019.559,-83.483,385.114,-24.015,21.647,-44.036
C08749=1019.558,-83.818,385.138,-24.015,21.648,-44.040
C08750=1019.555,-84.152,385.162,-24.014,21.648,-44.045
C08751=1019.554,-84.501,385.187,-24.013,21.649,-44.051
C08752=1019.551,-84.899,385.216,-24.012,21.650,-44.056
C08753=1019.550,-85.111,385.231,-24.012,21.649,-44.060
C08754=1019.550,-85.325,385.246,-24.012,21.649,-44.062
C08755=1019.548,-85.733,385.275,-24.011,21.650,-44.067
C08756=1019.545,-86.093,385.301,-24.010,21.651,-44.073
C08757=1019.544,-86.423,385.324,-24.009,21.652,-44.078
C08758=1019.542,-86.745,385.348,-24.009,21.652,-44.082
C08759=1019.540,-87.061,385.370,-24.008,21.653,-44.088
C08760=1019.538,-87.373,385.393,-24.007,21.653,-44.093
C08761=1019.537,-87.684,385.415,-24.007,21.654,-44.097
C08762=1019.535,-87.997,385.437,-24.006,21.654,-44.102
C08763=1019.533,-88.315,385.459,-24.006,21.655,-44.106
C08764=1019.531,-88.687,385.486,-24.005,21.656,-44.114
C08765=1019.530,-88.905,385.501,-24.004,21.656,-44.117
C08766=1019.528,-89.139,385.519,-24.004,21.656,-44.119
C08767=1019.527,-89.377,385.535,-24.004,21.656,-44.121
C08768=1019.526,-89.609,385.552,-24.004,21.657,-44.123
C08769=1019.523,-90.014,385.581,-24.003,21.658,-44.130
C08770=1019.522,-90.353,385.604,-24.002,21.658,-44.136
C08771=1019.519,-90.682,385.628,-24.001,21.659,-44.141
C08772=1019.518,-91.011,385.651,-24.001,21.660,-44.145
C08773=1019.515,-91.340,385.675,-24.000,21.660,-44.150
C08774=1019.513,-91.668,385.698,-23.999,21.660,-44.156
C08775=1019.511,-91.996,385.722,-23.999,21.661,-44.160
C08776=1019.509,-92.323,385.744,-23.998,21.662,-44.165
C08777=1019.507,-92.650,385.768,-23.998,21.662,-44.169
C08778=1019.505,-92.976,385.790,-23.997,21.663,-44.175
C08779=1019.503,-93.302,385.814,-23.996,21.663,-44.180
C08780=1019.501,-93.627,385.837,-23.996,21.664,-44.184
C08781=1019.499,-93.951,385.859,-23.995,21.664,-44.189
C08782=1019.497,-94.276,385.883,-23.994,21.665,-44.193
C08783=1019.495,-94.599,385.905,-23.994,21.666,-44.199
C08784=1019.493,-94.922,385.928,-23.993,21.666,-44.204
C08785=1019.490,-95.245,385.951,-23.993,21.666,-44.207
C08786=1019.489,-95.567,385.973,-23.992,21.667,-44.213
C08787=1019.487,-95.889,385.996,-23.991,21.668,-44.217
C08788=1019.484,-96.211,386.018,-23.991,21.668,-44.222
C08789=1019.482,-96.532,386.041,-23.990,21.669,-44.226
C08790=1019.479,-96.852,386.063,-23.989,21.669,-44.231
C08791=1019.478,-97.174,386.086,-23.989,21.670,-44.236
C08792=1019.476,-97.495,386.108,-23.988,21.670,-44.241
C08793=1019.473,-97.816,386.131,-23.987,21.670,-44.246
C08794=1019.471,-98.137,386.153,-23.987,21.672,-44.250
C08795=1019.469,-98.457,386.176,-23.986,21.671,-44.255
C08796=1019.466,-98.778,386.198,-23.986,21.673,-44.260
C08797=1019.464,-99.100,386.221,-23.985,21.673,-44.265
C08798=1019.461,-99.421,386.244,-23.985,21.673,-44.268
C08799=1019.459,-99.742,386.266,-23.984,21.674,-44.274
C08800=1019.457,-100.064,386.288,-23.983,21.675,-44.278
C08801=1019.455,-100.387,386.311,-23.983,21.675,-44.283
C08802=1019.452,-100.709,386.333,-23.982,21.676,-44.287
C08803=1019.450,-101.032,386.356,-23.981,21.676,-44.292
C08804=1019.448,-101.356,386.378,-23.981,21.677,-44.298
C08805=1019.445,-101.680,386.401,-23.980,21.677,-44.302
C08806=1019.443,-102.005,386.424,-23.980,21.678,-44.307
C08807=1019.440,-102.329,386.446,-23.979,21.679,-44.311
C08808=1019.437,-102.655,386.469,-23.978,21.679,-44.316
C08809=1019.435,-102.981,386.491,-23.978,21.680,-44.320
C08810=1019.432,-103.308,386.514,-23.977,21.680,-44.326
C08811=1019.430,-103.634,386.536,-23.976,21.681,-44.331
C08812=1019.427,-103.962,386.559,-23.976,21.681,-44.335
C08813=1019.425,-104.289,386.582,-23.975,21.681,-44.340
C08814=1019.422,-104.618,386.606,-23.975,21.683,-44.344
C08815=1019.419,-104.945,386.628,-23.974,21.683,-44.350
C08816=1019.416,-105.274,386.651,-23.974,21.684,-44.354
C08817=1019.414,-105.603,386.673,-23.973,21.684,-44.359
C08818=1019.411,-105.932,386.696,-23.972,21.685,-44.365
C08819=1019.408,-106.261,386.719,-23.972,21.685,-44.368
C08820=1019.406,-106.590,386.742,-23.971,21.685,-44.374
C08821=1019.403,-106.919,386.764,-23.971,21.687,-44.378
C08822=1019.400,-107.247,386.787,-23.970,21.687,-44.383
C08823=1019.398,-107.577,386.809,-23.969,21.687,-44.388
C08824=1019.395,-107.905,386.832,-23.969,21.688,-44.392
C08825=1019.392,-108.234,386.855,-23.968,21.689,-44.398
C08826=1019.389,-108.564,386.877,-23.967,21.689,-44.402
C08827=1019.387,-108.893,386.900,-23.967,21.689,-44.407
C08828=1019.384,-109.221,386.923,-23.966,21.690,-44.412
C08829=1019.381,-109.550,386.946,-23.965,21.691,-44.416
C08830=1019.378,-109.879,386.968,-23.965,21.691,-44.422
C08831=1019.375,-110.208,386.990,-23.964,21.692,-44.426
C08832=1019.372,-110.536,387.013,-23.963,21.692,-44.431
C08833=1019.369,-110.865,387.035,-23.963,21.693,-44.436
C08834=1019.366,-111.194,387.058,-23.962,21.693,-44.440
C08835=1019.363,-111.523,387.080,-23.962,21.694,-44.446
C08836=1019.360,-111.851,387.103,-23.961,21.695,-44.449
C08837=1019.357,-112.180,387.125,-23.960,21.695,-44.455
C08838=1019.354,-112.509,387.148,-23.960,21.696,-44.459
C08839=1019.351,-112.838,387.170,-23.959,21.696,-44.464
C08840=1019.348,-113.166,387.193,-23.958,21.697,-44.470
C08841=1019.345,-113.495,387.215,-23.958,21.697,-44.473
C08842=1019.342,-113.824,387.238,-23.957,21.698,-44.479
C08843=1019.339,-114.152,387.260,-23.957,21.699,-44.483
C08844=1019.336,-114.480,387.282,-23.956,21.699,-44.488
C08845=1019.333,-114.809,387.304,-23.956,21.700,-44.492
C08846=1019.330,-115.138,387.327,-23.955,21.700,-44.497
C08847=1019.327,-115.466,387.350,-23.954,21.701,-44.503
C08848=1019.324,-115.795,387.372,-23.954,21.701,-44.507
C08849=1019.321,-116.123,387.394,-23.953,21.701,-44.512
C08850=1019.318,-116.452,387.417,-23.953,21.703,-44.516
C08851=1019.314,-116.781,387.438,-23.952,21.703,-44.521
C08852=1019.311,-117.109,387.461,-23.951,21.704,-44.525
C08853=1019.308,-117.437,387.483,-23.951,21.704,-44.531
C08854=1019.305,-117.765,387.506,-23.950,21.705,-44.535
C08855=1019.301,-118.094,387.528,-23.949,21.705,-44.540
C08856=1019.298,-118.422,387.550,-23.949,21.705,-44.545
C08857=1019.294,-118.750,387.573,-23.948,21.707,-44.549
C08858=1019.292,-119.080,387.594,-23.948,21.707,-44.554
C08859=1019.288,-119.408,387.617,-23.947,21.707,-44.558
C08860=1019.285,-119.736,387.639,-23.946,21.708,-44.564
C08861=1019.282,-120.064,387.661,-23.946,21.709,-44.568
C08862=1019.278,-120.392,387.683,-23.945,21.709,-44.573
C08863=1019.275,-120.721,387.706,-23.945,21.710,-44.577
C08864=1019.271,-121.049,387.728,-23.944,21.710,-44.582
C08865=1019.268,-121.377,387.750,-23.944,21.711,-44.586
C08866=1019.264,-121.705,387.771,-23.943,21.711,-44.591
C08867=1019.261,-122.034,387.794,-23.942,21.712,-44.597
C08868=1019.257,-122.362,387.816,-23.942,21.713,-44.601
C08869=1019.254,-122.690,387.838,-23.941,21.713,-44.606
C08870=1019.251,-123.018,387.860,-23.940,21.714,-44.610
C08871=1019.247,-123.346,387.882,-23.940,21.714,-44.615
C08872=1019.243,-123.675,387.904,-23.939,21.715,-44.620
C08873=1019.239,-124.003,387.926,-23.939,21.715,-44.625
C08874=1019.236,-124.331,387.949,-23.938,21.716,-44.628
C08875=1019.233,-124.659,387.970,-23.937,21.717,-44.634
C08876=1019.229,-124.987,387.993,-23.937,21.717,-44.638
C08877=1019.225,-125.315,388.015,-23.936,21.717,-44.643
C08878=1019.222,-125.644,388.036,-23.936,21.719,-44.647
C08879=1019.218,-125.971,388.057,-23.935,21.719,-44.652
C08880=1019.214,-126.300,388.079,-23.935,21.720,-44.657
C08881=1019.211,-126.628,388.101,-23.934,21.720,-44.662
C08882=1019.207,-126.956,388.123,-23.933,21.720,-44.667
C08883=1019.204,-127.284,388.145,-23.933,21.721,-44.671
C08884=1019.200,-127.612,388.167,-23.932,21.721,-44.676
C08885=1019.196,-127.940,388.189,-23.931,21.722,-44.680
C08886=1019.192,-128.269,388.211,-23.931,21.723,-44.686
C08887=1019.188,-128.596,388.233,-23.930,21.723,-44.689
C08888=1019.185,-128.924,388.255,-23.929,21.723,-44.695
C08889=1019.181,-129.252,388.277,-23.929,21.725,-44.699
C08890=1019.176,-129.580,388.298,-23.928,21.724,-44.704
C08891=1019.173,-129.908,388.320,-23.928,21.726,-44.708
C08892=1019.169,-130.236,388.342,-23.927,21.726,-44.713
C08893=1019.165,-130.564,388.364,-23.927,21.726,-44.717
C08894=1019.161,-130.892,388.386,-23.926,21.727,-44.723
C08895=1019.157,-131.220,388.408,-23.926,21.728,-44.726
C08896=1019.153,-131.548,388.429,-23.925,21.728,-44.732
C08897=1019.150,-131.876,388.451,-23.924,21.729,-44.736
C08898=1019.145,-132.204,388.473,-23.924,21.729,-44.741
C08899=1019.141,-132.532,388.495,-23.923,21.730,-44.745
C08900=1019.137,-132.860,388.516,-23.922,21.731,-44.750
C08901=1019.134,-133.188,388.538,-23.922,21.731,-44.754
C08902=1019.129,-133.516,388.559,-23.921,21.731,-44.759
C08903=1019.126,-133.844,388.581,-23.921,21.732,-44.763
C08904=1019.502,-133.817,388.347,-23.921,21.732,-44.763
C08905=1019.506,-133.489,388.324,-23.921,21.731,-44.759
C08906=1019.510,-133.161,388.303,-23.922,21.731,-44.754
C08907=1019.513,-132.833,388.281,-23.922,21.731,-44.750
C08908=1019.518,-132.505,388.260,-23.923,21.730,-44.745
C08909=1019.522,-132.177,388.238,-23.924,21.729,-44.741
C08910=1019.526,-131.850,388.216,-23.924,21.729,-44.736
C08911=1019.529,-131.521,388.194,-23.925,21.728,-44.732
C08912=1019.533,-131.193,388.173,-23.926,21.728,-44.726
C08913=1019.537,-130.865,388.152,-23.926,21.727,-44.723
C08914=1019.540,-130.537,388.130,-23.927,21.726,-44.717
C08915=1019.545,-130.209,388.108,-23.927,21.726,-44.713
C08916=1019.549,-129.881,388.086,-23.928,21.726,-44.708
C08917=1019.552,-129.553,388.064,-23.928,21.724,-44.704
C08918=1019.556,-129.225,388.042,-23.929,21.725,-44.699
C08919=1019.560,-128.897,388.021,-23.929,21.723,-44.695
C08920=1019.563,-128.570,387.999,-23.930,21.723,-44.689
C08921=1019.567,-128.241,387.977,-23.931,21.723,-44.686
C08922=1019.571,-127.913,387.955,-23.931,21.722,-44.680
C08923=1019.575,-127.585,387.933,-23.932,21.721,-44.676
C08924=1019.578,-127.257,387.912,-23.933,21.721,-44.671
C08925=1019.582,-126.929,387.890,-23.933,21.720,-44.667
C08926=1019.586,-126.600,387.868,-23.934,21.720,-44.662
C08927=1019.589,-126.273,387.846,-23.935,21.720,-44.657
C08928=1019.593,-125.945,387.824,-23.935,21.719,-44.652
C08929=1019.597,-125.616,387.802,-23.936,21.719,-44.647
C08930=1019.600,-125.288,387.780,-23.936,21.717,-44.643
C08931=1019.604,-124.961,387.758,-23.937,21.717,-44.638
C08932=1019.607,-124.632,387.736,-23.937,21.717,-44.634
C08933=1019.611,-124.304,387.714,-23.938,21.716,-44.628
C08934=1019.615,-123.975,387.693,-23.939,21.715,-44.625
C08935=1019.618,-123.648,387.671,-23.939,21.715,-44.620
C08936=1019.622,-123.319,387.649,-23.940,21.714,-44.615
C08937=1019.625,-122.991,387.626,-23.940,21.714,-44.610
C08938=1019.628,-122.663,387.604,-23.941,21.713,-44.606
C08939=1019.631,-122.335,387.582,-23.942,21.713,-44.601
C08940=1019.635,-122.007,387.560,-23.942,21.712,-44.597
C08941=1019.639,-121.679,387.538,-23.943,21.711,-44.591
C08942=1019.642,-121.349,387.516,-23.944,21.711,-44.586
C08943=1019.645,-121.022,387.494,-23.944,21.710,-44.582
C08944=1019.649,-120.694,387.472,-23.945,21.710,-44.577
C08945=1019.652,-120.365,387.450,-23.945,21.709,-44.573
C08946=1019.656,-120.037,387.428,-23.946,21.709,-44.568
C08947=1019.659,-119.709,387.406,-23.946,21.708,-44.564
C08948=1019.661,-119.380,387.384,-23.947,21.707,-44.558
C08949=1019.665,-119.052,387.362,-23.948,21.707,-44.554
C08950=1019.668,-118.723,387.339,-23.948,21.707,-44.549
C08951=1019.672,-118.395,387.317,-23.949,21.705,-44.545
C08952=1019.674,-118.067,387.295,-23.949,21.705,-44.540
C08953=1019.678,-117.739,387.273,-23.950,21.705,-44.535
C08954=1019.681,-117.410,387.251,-23.951,21.704,-44.531
C08955=1019.685,-117.081,387.228,-23.951,21.704,-44.525
C08956=1019.688,-116.753,387.206,-23.952,21.703,-44.521
C08957=1019.691,-116.425,387.184,-23.953,21.703,-44.516
C08958=1019.694,-116.097,387.161,-23.953,21.701,-44.512
C08959=1019.697,-115.767,387.139,-23.954,21.701,-44.507
C08960=1019.700,-115.439,387.117,-23.954,21.701,-44.503
C08961=1019.703,-115.111,387.095,-23.955,21.700,-44.497
C08962=1019.707,-114.782,387.072,-23.956,21.700,-44.492
C08963=1019.710,-114.454,387.049,-23.956,21.699,-44.488
C08964=1019.712,-114.125,387.028,-23.957,21.699,-44.483
C08965=1019.715,-113.797,387.005,-23.957,21.698,-44.479
C08966=1019.718,-113.468,386.983,-23.958,21.697,-44.473
C08967=1019.722,-113.140,386.960,-23.958,21.697,-44.470
C08968=1019.724,-112.810,386.938,-23.959,21.696,-44.464
C08969=1019.727,-112.482,386.915,-23.960,21.696,-44.459
C08970=1019.730,-112.153,386.893,-23.960,21.695,-44.455
C08971=1019.733,-111.824,386.871,-23.961,21.695,-44.449
C08972=1019.736,-111.496,386.848,-23.962,21.694,-44.446
C08973=1019.739,-111.167,386.825,-23.962,21.693,-44.440
C08974=1019.742,-110.838,386.803,-23.963,21.693,-44.436
C08975=1019.745,-110.509,386.781,-23.963,21.692,-44.431
C08976=1019.748,-110.181,386.758,-23.964,21.692,-44.426
C08977=1019.751,-109.852,386.735,-23.965,21.691,-44.422
C08978=1019.754,-109.523,386.713,-23.965,21.691,-44.416
C08979=1019.756,-109.194,386.690,-23.966,21.690,-44.412
C08980=1019.759,-108.865,386.667,-23.967,21.689,-44.407
C08981=1019.762,-108.536,386.645,-23.967,21.689,-44.402
C08982=1019.765,-108.208,386.623,-23.968,21.689,-44.398
C08983=1019.767,-107.878,386.600,-23.969,21.688,-44.392
C08984=1019.770,-107.550,386.577,-23.969,21.687,-44.388
C08985=1019.773,-107.221,386.555,-23.970,21.687,-44.383
C08986=1019.775,-106.891,386.532,-23.971,21.687,-44.378
C08987=1019.778,-106.563,386.509,-23.971,21.685,-44.374
C08988=1019.781,-106.234,386.487,-23.972,21.685,-44.368
C08989=1019.783,-105.905,386.464,-23.972,21.685,-44.365
C08990=1019.786,-105.576,386.441,-23.973,21.684,-44.359
C08991=1019.789,-105.248,386.419,-23.974,21.684,-44.354
C08992=1019.791,-104.919,386.395,-23.974,21.683,-44.350
C08993=1019.794,-104.591,386.373,-23.975,21.683,-44.344
C08994=1019.797,-104.262,386.350,-23.975,21.681,-44.340
C08995=1019.799,-103.935,386.328,-23.976,21.681,-44.335
C08996=1019.802,-103.607,386.305,-23.976,21.681,-44.331
C08997=1019.804,-103.281,386.282,-23.977,21.680,-44.326
C08998=1019.806,-102.954,386.260,-23.978,21.680,-44.320
C08999=1019.809,-102.628,386.238,-23.978,21.679,-44.316
C09000=1019.812,-102.302,386.214,-23.979,21.679,-44.311
C09001=1019.814,-101.977,386.192,-23.980,21.678,-44.307
C09002=1019.816,-101.653,386.170,-23.980,21.677,-44.302
C09003=1019.819,-101.329,386.146,-23.981,21.677,-44.298
C09004=1019.821,-101.005,386.124,-23.981,21.676,-44.292
C09005=1019.823,-100.683,386.101,-23.982,21.676,-44.287
C09006=1019.826,-100.359,386.079,-23.983,21.675,-44.283
C09007=1019.829,-100.038,386.057,-23.983,21.675,-44.278
C09008=1019.830,-99.715,386.035,-23.984,21.674,-44.274
C09009=1019.833,-99.394,386.012,-23.985,21.673,-44.268
C09010=1019.835,-99.073,385.989,-23.985,21.673,-44.265
C09011=1019.837,-98.752,385.967,-23.986,21.673,-44.260
C09012=1019.839,-98.431,385.945,-23.986,21.671,-44.255
C09013=1019.842,-98.110,385.922,-23.987,21.672,-44.250
C09014=1019.844,-97.789,385.900,-23.987,21.670,-44.246
C09015=1019.846,-97.468,385.878,-23.988,21.670,-44.241
C09016=1019.849,-97.147,385.855,-23.989,21.670,-44.236
C09017=1019.851,-96.826,385.833,-23.989,21.669,-44.231
C09018=1019.852,-96.505,385.810,-23.990,21.669,-44.226
C09019=1019.855,-96.184,385.787,-23.991,21.668,-44.222
C09020=1019.857,-95.862,385.764,-23.991,21.668,-44.217
C09021=1019.859,-95.539,385.742,-23.992,21.667,-44.213
C09022=1019.862,-95.218,385.719,-23.993,21.666,-44.207
C09023=1019.864,-94.895,385.696,-23.993,21.666,-44.204
C09024=1019.866,-94.573,385.674,-23.994,21.666,-44.199
C09025=1019.868,-94.249,385.651,-23.994,21.665,-44.193
C09026=1019.870,-93.924,385.628,-23.995,21.664,-44.189
C09027=1019.872,-93.600,385.605,-23.996,21.664,-44.184
C09028=1019.874,-93.275,385.582,-23.996,21.663,-44.180
C09029=1019.876,-92.949,385.560,-23.997,21.663,-44.175
C09030=1019.878,-92.624,385.537,-23.998,21.662,-44.169
C09031=1019.880,-92.296,385.513,-23.998,21.662,-44.165
C09032=1019.882,-91.969,385.490,-23.999,21.661,-44.160
C09033=1019.884,-91.641,385.467,-23.999,21.660,-44.156
C09034=1019.886,-91.313,385.443,-24.000,21.660,-44.150
C09035=1019.888,-90.985,385.420,-24.001,21.660,-44.145
C09036=1019.889,-90.655,385.397,-24.001,21.659,-44.141
C09037=1019.892,-90.325,385.374,-24.002,21.658,-44.136
C09038=1019.894,-89.988,385.349,-24.003,21.658,-44.130
C09039=1019.896,-89.582,385.321,-24.004,21.657,-44.123
C09040=1019.897,-89.351,385.305,-24.004,21.656,-44.121
C09041=1019.899,-89.112,385.288,-24.004,21.656,-44.119
C09042=1019.900,-88.879,385.271,-24.004,21.656,-44.117
C09043=1019.902,-88.463,385.242,-24.005,21.656,-44.110
C09044=1019.904,-88.288,385.228,-24.006,21.655,-44.106
C09045=1019.905,-87.970,385.206,-24.006,21.654,-44.102
C09046=1019.907,-87.657,385.184,-24.007,21.654,-44.097
C09047=1019.909,-87.346,385.162,-24.007,21.653,-44.093
C09048=1019.910,-87.034,385.139,-24.008,21.653,-44.088
C09049=1019.912,-86.718,385.117,-24.009,21.652,-44.082
C09050=1019.914,-86.395,385.094,-24.009,21.652,-44.078
C09051=1019.916,-86.066,385.070,-24.010,21.651,-44.073
C09052=1019.918,-85.707,385.045,-24.011,21.650,-44.067
C09053=1019.920,-85.298,385.015,-24.012,21.649,-44.062
C09054=1019.920,-85.084,385.000,-24.012,21.649,-44.060
C09055=1019.922,-84.872,384.985,-24.012,21.650,-44.056
C09056=1019.924,-84.475,384.956,-24.013,21.649,-44.051
C09057=1019.925,-84.125,384.931,-24.014,21.648,-44.045
C09058=1019.928,-83.791,384.908,-24.015,21.648,-44.040
C09059=1019.929,-83.456,384.883,-24.015,21.647,-44.036
C09060=1019.930,-83.121,384.860,-24.016,21.647,-44.031
C09061=1019.932,-82.785,384.836,-24.016,21.646,-44.025
C09062=1019.933,-82.449,384.811,-24.017,21.645,-44.021
C09063=1019.936,-82.113,384.786,-24.018,21.645,-44.016
C09064=1019.937,-81.776,384.763,-24.018,21.645,-44.010
C09065=1019.939,-81.439,384.738,-24.019,21.644,-44.005
C09066=1019.940,-81.101,384.715,-24.020,21.643,-44.001
C09067=1019.941,-80.762,384.689,-24.020,21.643,-43.995
C09068=1019.943,-80.424,384.665,-24.021,21.643,-43.990
C09069=1019.945,-80.085,384.641,-24.021,21.641,-43.986
C09070=1019.947,-79.745,384.616,-24.022,21.641,-43.981
C09071=1019.948,-79.406,384.591,-24.023,21.641,-43.975
C09072=1019.949,-79.065,384.567,-24.023,21.639,-43.971
C09073=1019.951,-78.725,384.542,-24.024,21.639,-43.966
C09074=1019.952,-78.384,384.518,-24.025,21.638,-43.960
C09075=1019.954,-78.043,384.493,-24.026,21.639,-43.955
C09076=1019.955,-77.701,384.468,-24.026,21.637,-43.951
C09077=1019.957,-77.360,384.443,-24.027,21.637,-43.946
C09078=1019.958,-77.019,384.418,-24.028,21.636,-43.940
C09079=1019.960,-76.676,384.393,-24.028,21.636,-43.936
C09080=1019.961,-76.333,384.369,-24.029,21.635,-43.931
C09081=1019.962,-75.991,384.343,-24.030,21.635,-43.926
C09082=1019.963,-75.648,384.319,-24.030,21.634,-43.920
C09083=1019.965,-75.305,384.293,-24.031,21.634,-43.916
C09084=1019.967,-74.962,384.269,-24.031,21.633,-43.911
C09085=1019.967,-74.618,384.243,-24.032,21.633,-43.905
C09086=1019.969,-74.275,384.218,-24.033,21.632,-43.901
C09087=1019.970,-73.931,384.194,-24.033,21.632,-43.896
C09088=1019.972,-73.587,384.168,-24.034,21.631,-43.890
C09089=1019.972,-73.244,384.143,-24.035,21.630,-43.885
C09090=1019.974,-72.900,384.118,-24.035,21.630,-43.881
C09091=1019.975,-72.556,384.093,-24.036,21.629,-43.875
C09092=1019.977,-72.212,384.068,-24.037,21.629,-43.870
C09093=1019.978,-71.868,384.043,-24.038,21.628,-43.865
C09094=1019.979,-71.524,384.018,-24.038,21.628,-43.861
C09095=1019.980,-71.180,383.992,-24.039,21.627,-43.855
C09096=1019.981,-70.836,383.966,-24.040,21.627,-43.850
C09097=1019.983,-70.492,383.942,-24.040,21.626,-43.844
C09098=1019.983,-70.149,383.916,-24.041,21.625,-43.840
C09099=1019.984,-69.804,383.891,-24.041,21.625,-43.835
C09100=1019.986,-69.460,383.865,-24.042,21.624,-43.829
C09101=1019.987,-69.115,383.840,-24.043,21.624,-43.824
C09102=1019.987,-68.772,383.815,-24.043,21.623,-43.820
C09103=1019.988,-68.428,383.789,-24.044,21.623,-43.815
C09104=1019.990,-68.085,383.764,-24.045,21.622,-43.809
C09105=1019.991,-67.741,383.739,-24.045,21.622,-43.805
C09106=1019.991,-67.398,383.714,-24.046,21.621,-43.800
C09107=1019.993,-67.054,383.688,-24.047,21.621,-43.795
C09108=1019.994,-66.711,383.663,-24.048,21.620,-43.789
C09109=1019.995,-66.368,383.637,-24.048,21.620,-43.785
C09110=1019.996,-66.025,383.612,-24.049,21.619,-43.780
C09111=1019.997,-65.683,383.587,-24.050,21.619,-43.774
C09112=1019.997,-65.340,383.561,-24.050,21.617,-43.770
C09113=1019.999,-64.998,383.536,-24.051,21.618,-43.765
C09114=1019.999,-64.657,383.510,-24.051,21.617,-43.759
C09115=1020.000,-64.315,383.485,-24.052,21.617,-43.754
C09116=1020.001,-63.973,383.460,-24.053,21.615,-43.750
C09117=1020.002,-63.633,383.435,-24.053,21.616,-43.745
C09118=1020.003,-63.292,383.409,-24.054,21.615,-43.739
C09119=1020.004,-62.951,383.384,-24.055,21.614,-43.735
C09120=1020.004,-62.612,383.359,-24.055,21.613,-43.730
C09121=1020.005,-62.272,383.333,-24.056,21.614,-43.725
C09122=1020.006,-61.933,383.308,-24.057,21.612,-43.720
C09123=1020.007,-61.594,383.282,-24.057,21.612,-43.715
C09124=1020.007,-61.256,383.257,-24.058,21.611,-43.710
C09125=1020.009,-60.918,383.232,-24.059,21.611,-43.706
